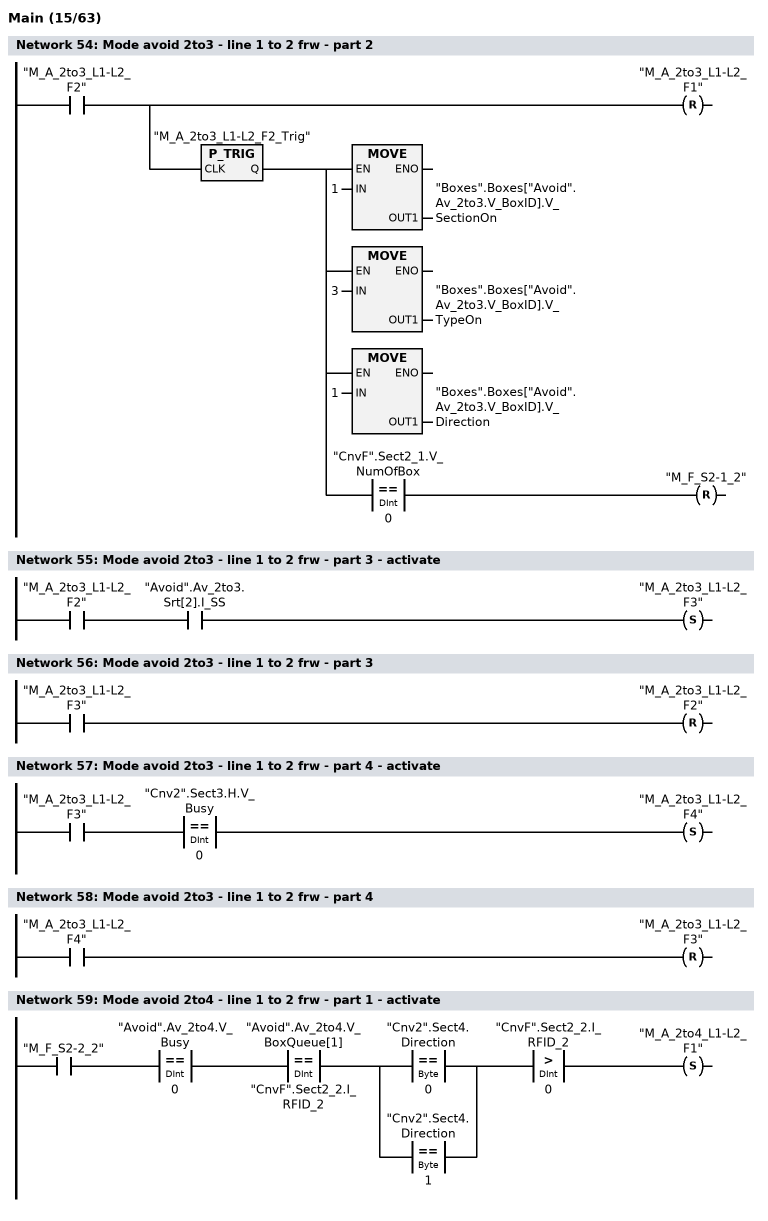
   RUNG wire#powerrail
      Contact( "M_A_2to3_L1-L2_F2" )
      wire#w1
      R_Coil( "M_A_2to3_L1-L2_F1" )
   END_RUNG
   RUNG wire#w1
      P_Trig( "M_A_2to3_L1-L2_F2_Trig" )
      wire#w2
      Move(in := 1, out1 => "Boxes".Boxes["Avoid".Av_2to3.V_BoxID].V_SectionOn)
   END_RUNG
   RUNG wire#w2
      Move(in := 3, out1 => "Boxes".Boxes["Avoid".Av_2to3.V_BoxID].V_TypeOn)
   END_RUNG
   RUNG wire#w2
      Move(in := 1, out1 => "Boxes".Boxes["Avoid".Av_2to3.V_BoxID].V_Direction)
   END_RUNG
   RUNG wire#w2
      { S7_Templates := "SrcType := DInt" } EQ_Contact(in1 := "CnvF".Sect2_1.V_NumOfBox, in2 := 0)
      R_Coil( "M_F_S2-1_2" )
   END_RUNG
   // the same network as SCL:
   IF "M_A_2to3_L1-L2_F2" THEN "M_A_2to3_L1-L2_F1" := FALSE; END_IF;
   #_w1 := "M_A_2to3_L1-L2_F2" AND NOT "M_A_2to3_L1-L2_F2_Trig";   // rising edge
   "M_A_2to3_L1-L2_F2_Trig" := "M_A_2to3_L1-L2_F2";
   IF #_w1 THEN
       "Boxes".Boxes["Avoid".Av_2to3.V_BoxID].V_SectionOn := 1;
       "Boxes".Boxes["Avoid".Av_2to3.V_BoxID].V_TypeOn := 3;
       "Boxes".Boxes["Avoid".Av_2to3.V_BoxID].V_Direction := 1;
   END_IF;
   IF #_w1 AND ("CnvF".Sect2_1.V_NumOfBox = 0) THEN "M_F_S2-1_2" := FALSE; END_IF;
END_REGION

REGION Network 55: Mode avoid 2to3 - line 1 to 2 frw - part 3 - activate
   RUNG wire#powerrail
      Contact( "M_A_2to3_L1-L2_F2" )
      Contact( "Avoid".Av_2to3.Srt[2].I_SS )
      S_Coil( "M_A_2to3_L1-L2_F3" )
   END_RUNG
   // the same network as SCL:
   IF "M_A_2to3_L1-L2_F2" AND "Avoid".Av_2to3.Srt[2].I_SS THEN "M_A_2to3_L1-L2_F3" := TRUE; END_IF;
END_REGION

REGION Network 56: Mode avoid 2to3 - line 1 to 2 frw - part 3
   RUNG wire#powerrail
      Contact( "M_A_2to3_L1-L2_F3" )
      R_Coil( "M_A_2to3_L1-L2_F2" )
   END_RUNG
   // the same network as SCL:
   IF "M_A_2to3_L1-L2_F3" THEN "M_A_2to3_L1-L2_F2" := FALSE; END_IF;
END_REGION

REGION Network 57: Mode avoid 2to3 - line 1 to 2 frw - part 4 - activate
   RUNG wire#powerrail
      Contact( "M_A_2to3_L1-L2_F3" )
      { S7_Templates := "SrcType := DInt" } EQ_Contact(in1 := "Cnv2".Sect3.H.V_Busy, in2 := 0)
      S_Coil( "M_A_2to3_L1-L2_F4" )
   END_RUNG
   // the same network as SCL:
   IF "M_A_2to3_L1-L2_F3" AND ("Cnv2".Sect3.H.V_Busy = 0) THEN "M_A_2to3_L1-L2_F4" := TRUE; END_IF;
END_REGION

REGION Network 58: Mode avoid 2to3 - line 1 to 2 frw - part 4
   RUNG wire#powerrail
      Contact( "M_A_2to3_L1-L2_F4" )
      R_Coil( "M_A_2to3_L1-L2_F3" )
   END_RUNG
   // the same network as SCL:
   IF "M_A_2to3_L1-L2_F4" THEN "M_A_2to3_L1-L2_F3" := FALSE; END_IF;
END_REGION

REGION Network 59: Mode avoid 2to4 - line 1 to 2 frw - part 1 - activate
   RUNG wire#powerrail
      Contact( "M_F_S2-2_2" )
      { S7_Templates := "SrcType := DInt" } EQ_Contact(in1 := "Avoid".Av_2to4.V_Busy, in2 := 0)
      { S7_Templates := "SrcType := DInt" } EQ_Contact(in1 := "Avoid".Av_2to4.V_BoxQueue[1], in2 := "CnvF".Sect2_2.I_RFID_2)
      wire#w1
      { S7_Templates := "SrcType := Byte" } EQ_Contact(in1 := "Cnv2".Sect4.Direction, in2 := 0)
      wire#w2
      { S7_Templates := "SrcType := DInt" } GT_Contact(in1 := "CnvF".Sect2_2.I_RFID_2, in2 := 0)
      S_Coil( "M_A_2to4_L1-L2_F1" )
   END_RUNG
   RUNG wire#w1
      { S7_Templates := "SrcType := Byte" } EQ_Contact(in1 := "Cnv2".Sect4.Direction, in2 := 1)
   END_RUNG wire#w2
   // the same network as SCL:
   IF "M_F_S2-2_2" AND ("Avoid".Av_2to4.V_Busy = 0) AND ("Avoid".Av_2to4.V_BoxQueue[1] = "CnvF".Sect2_2.I_RFID_2) AND (("Cnv2".Sect4.Direction = 0) OR ("Cnv2".Sect4.Direction = 1)) AND ("CnvF".Sect2_2.I_RFID_2 > 0) THEN
       "M_A_2to4_L1-L2_F1" := TRUE;
   END_IF;
END_REGION

REGION Network 60: Mode avoid 2to4 - line 1 to 2 frw - part 1
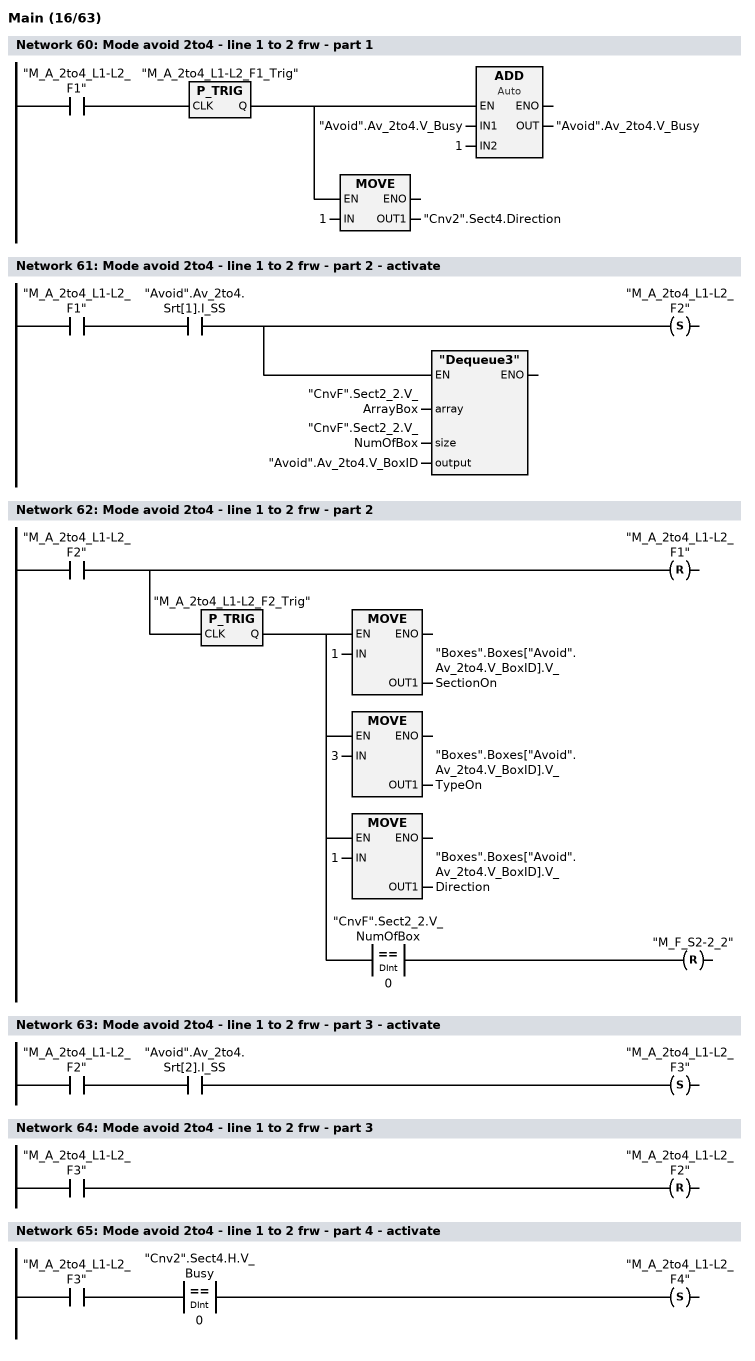
   RUNG wire#powerrail
      Contact( "M_A_2to4_L1-L2_F1" )
      P_Trig( "M_A_2to4_L1-L2_F1_Trig" )
      wire#w1
      Add(in1 := "Avoid".Av_2to4.V_Busy, in2 := 1, out => "Avoid".Av_2to4.V_Busy)
   END_RUNG
   RUNG wire#w1
      Move(in := 1, out1 => "Cnv2".Sect4.Direction)
   END_RUNG
   // the same network as SCL:
   #_w1 := "M_A_2to4_L1-L2_F1" AND NOT "M_A_2to4_L1-L2_F1_Trig";   // rising edge
   "M_A_2to4_L1-L2_F1_Trig" := "M_A_2to4_L1-L2_F1";
   IF #_w1 THEN
       "Avoid".Av_2to4.V_Busy := "Avoid".Av_2to4.V_Busy + 1;
       "Cnv2".Sect4.Direction := 1;
   END_IF;
END_REGION

REGION Network 61: Mode avoid 2to4 - line 1 to 2 frw - part 2 - activate
   RUNG wire#powerrail
      Contact( "M_A_2to4_L1-L2_F1" )
      Contact( "Avoid".Av_2to4.Srt[1].I_SS )
      wire#w1
      S_Coil( "M_A_2to4_L1-L2_F2" )
   END_RUNG
   RUNG wire#w1
      "Dequeue3"("array" := "CnvF".Sect2_2.V_ArrayBox, size := "CnvF".Sect2_2.V_NumOfBox, output := "Avoid".Av_2to4.V_BoxID)
   END_RUNG
   // the same network as SCL:
   IF "M_A_2to4_L1-L2_F1" AND "Avoid".Av_2to4.Srt[1].I_SS THEN
       "M_A_2to4_L1-L2_F2" := TRUE;
       "Dequeue3"("array" := "CnvF".Sect2_2.V_ArrayBox,
                  size := "CnvF".Sect2_2.V_NumOfBox,
                  output := "Avoid".Av_2to4.V_BoxID);
   END_IF;
END_REGION

REGION Network 62: Mode avoid 2to4 - line 1 to 2 frw - part 2
   RUNG wire#powerrail
      Contact( "M_A_2to4_L1-L2_F2" )
      wire#w1
      R_Coil( "M_A_2to4_L1-L2_F1" )
   END_RUNG
   RUNG wire#w1
      P_Trig( "M_A_2to4_L1-L2_F2_Trig" )
      wire#w2
      Move(in := 1, out1 => "Boxes".Boxes["Avoid".Av_2to4.V_BoxID].V_SectionOn)
   END_RUNG
   RUNG wire#w2
      Move(in := 3, out1 => "Boxes".Boxes["Avoid".Av_2to4.V_BoxID].V_TypeOn)
   END_RUNG
   RUNG wire#w2
      Move(in := 1, out1 => "Boxes".Boxes["Avoid".Av_2to4.V_BoxID].V_Direction)
   END_RUNG
   RUNG wire#w2
      { S7_Templates := "SrcType := DInt" } EQ_Contact(in1 := "CnvF".Sect2_2.V_NumOfBox, in2 := 0)
      R_Coil( "M_F_S2-2_2" )
   END_RUNG
   // the same network as SCL:
   IF "M_A_2to4_L1-L2_F2" THEN "M_A_2to4_L1-L2_F1" := FALSE; END_IF;
   #_w1 := "M_A_2to4_L1-L2_F2" AND NOT "M_A_2to4_L1-L2_F2_Trig";   // rising edge
   "M_A_2to4_L1-L2_F2_Trig" := "M_A_2to4_L1-L2_F2";
   IF #_w1 THEN
       "Boxes".Boxes["Avoid".Av_2to4.V_BoxID].V_SectionOn := 1;
       "Boxes".Boxes["Avoid".Av_2to4.V_BoxID].V_TypeOn := 3;
       "Boxes".Boxes["Avoid".Av_2to4.V_BoxID].V_Direction := 1;
   END_IF;
   IF #_w1 AND ("CnvF".Sect2_2.V_NumOfBox = 0) THEN "M_F_S2-2_2" := FALSE; END_IF;
END_REGION

REGION Network 63: Mode avoid 2to4 - line 1 to 2 frw - part 3 - activate
   RUNG wire#powerrail
      Contact( "M_A_2to4_L1-L2_F2" )
      Contact( "Avoid".Av_2to4.Srt[2].I_SS )
      S_Coil( "M_A_2to4_L1-L2_F3" )
   END_RUNG
   // the same network as SCL:
   IF "M_A_2to4_L1-L2_F2" AND "Avoid".Av_2to4.Srt[2].I_SS THEN "M_A_2to4_L1-L2_F3" := TRUE; END_IF;
END_REGION

REGION Network 64: Mode avoid 2to4 - line 1 to 2 frw - part 3
   RUNG wire#powerrail
      Contact( "M_A_2to4_L1-L2_F3" )
      R_Coil( "M_A_2to4_L1-L2_F2" )
   END_RUNG
   // the same network as SCL:
   IF "M_A_2to4_L1-L2_F3" THEN "M_A_2to4_L1-L2_F2" := FALSE; END_IF;
END_REGION

REGION Network 65: Mode avoid 2to4 - line 1 to 2 frw - part 4 - activate
   RUNG wire#powerrail
      Contact( "M_A_2to4_L1-L2_F3" )
      { S7_Templates := "SrcType := DInt" } EQ_Contact(in1 := "Cnv2".Sect4.H.V_Busy, in2 := 0)
      S_Coil( "M_A_2to4_L1-L2_F4" )
   END_RUNG
   // the same network as SCL:
   IF "M_A_2to4_L1-L2_F3" AND ("Cnv2".Sect4.H.V_Busy = 0) THEN "M_A_2to4_L1-L2_F4" := TRUE; END_IF;
END_REGION

REGION Network 66: Mode avoid 2to4 - line 1 to 2 frw - part 4
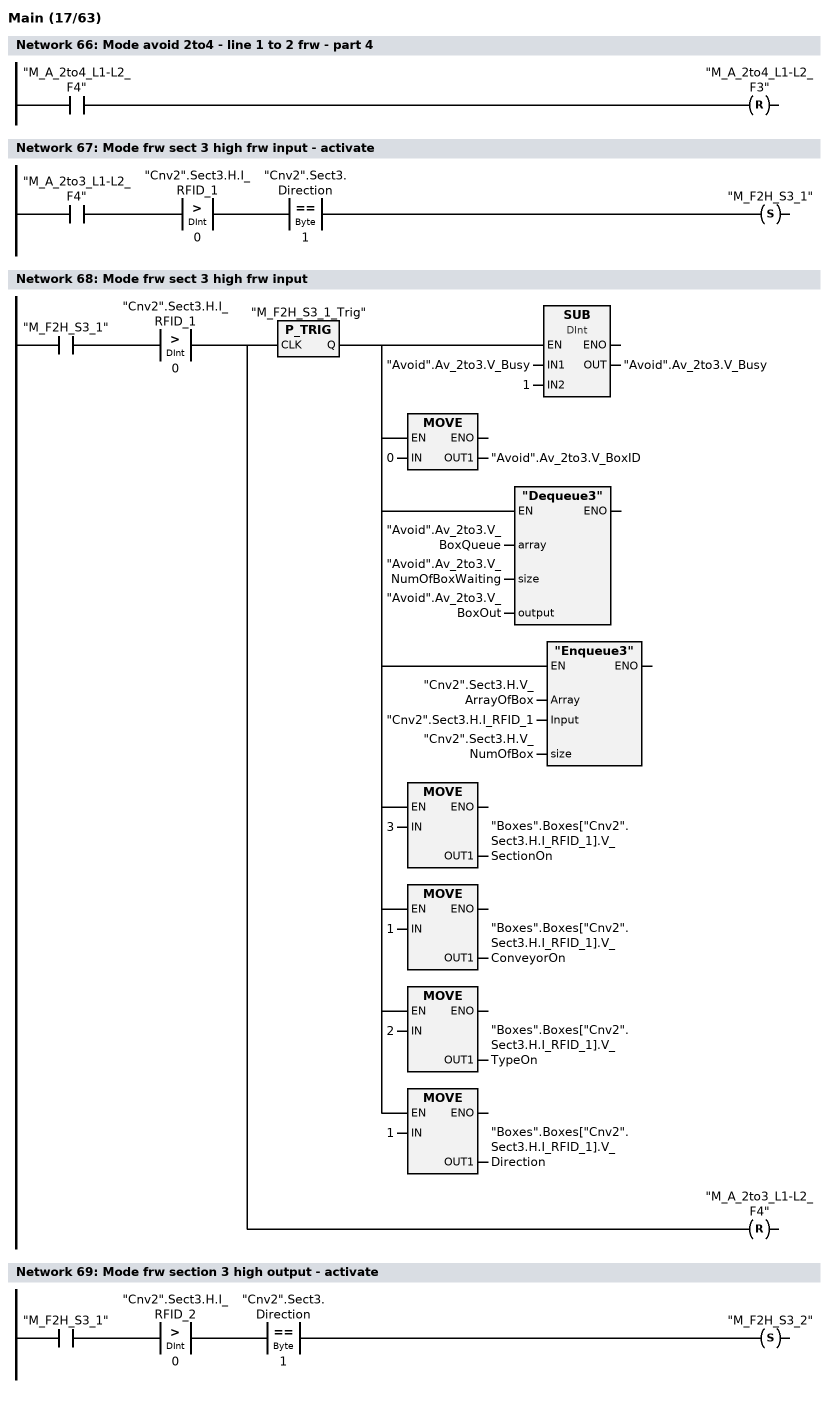
   RUNG wire#powerrail
      Contact( "M_A_2to4_L1-L2_F4" )
      R_Coil( "M_A_2to4_L1-L2_F3" )
   END_RUNG
   // the same network as SCL:
   IF "M_A_2to4_L1-L2_F4" THEN "M_A_2to4_L1-L2_F3" := FALSE; END_IF;
END_REGION

REGION Network 67: Mode frw sect 3 high frw input - activate
   RUNG wire#powerrail
      Contact( "M_A_2to3_L1-L2_F4" )
      { S7_Templates := "SrcType := DInt" } GT_Contact(in1 := "Cnv2".Sect3.H.I_RFID_1, in2 := 0)
      { S7_Templates := "SrcType := Byte" } EQ_Contact(in1 := "Cnv2".Sect3.Direction, in2 := 1)
      S_Coil( "M_F2H_S3_1" )
   END_RUNG
   // the same network as SCL:
   IF "M_A_2to3_L1-L2_F4" AND ("Cnv2".Sect3.H.I_RFID_1 > 0) AND ("Cnv2".Sect3.Direction = 1) THEN
       "M_F2H_S3_1" := TRUE;
   END_IF;
END_REGION

REGION Network 68: Mode frw sect 3 high frw input
   RUNG wire#powerrail
      Contact( "M_F2H_S3_1" )
      { S7_Templates := "SrcType := DInt" } GT_Contact(in1 := "Cnv2".Sect3.H.I_RFID_1, in2 := 0)
      wire#w1
      P_Trig( "M_F2H_S3_1_Trig" )
      wire#w2
      { S7_Templates := "SrcType := DInt" } Sub(in1 := "Avoid".Av_2to3.V_Busy, in2 := 1, out => "Avoid".Av_2to3.V_Busy)
   END_RUNG
   RUNG wire#w2
      Move(in := 0, out1 => "Avoid".Av_2to3.V_BoxID)
   END_RUNG
   RUNG wire#w2
      "Dequeue3"("array" := "Avoid".Av_2to3.V_BoxQueue, size := "Avoid".Av_2to3.V_NumOfBoxWaiting, output := "Avoid".Av_2to3.V_BoxOut)
   END_RUNG
   RUNG wire#w2
      "Enqueue3"("Array" := "Cnv2".Sect3.H.V_ArrayOfBox, Input := "Cnv2".Sect3.H.I_RFID_1, size := "Cnv2".Sect3.H.V_NumOfBox)
   END_RUNG
   RUNG wire#w2
      Move(in := 3, out1 => "Boxes".Boxes["Cnv2".Sect3.H.I_RFID_1].V_SectionOn)
   END_RUNG
   RUNG wire#w2
      Move(in := 1, out1 => "Boxes".Boxes["Cnv2".Sect3.H.I_RFID_1].V_ConveyorOn)
   END_RUNG
   RUNG wire#w2
      Move(in := 2, out1 => "Boxes".Boxes["Cnv2".Sect3.H.I_RFID_1].V_TypeOn)
   END_RUNG
   RUNG wire#w2
      Move(in := 1, out1 => "Boxes".Boxes["Cnv2".Sect3.H.I_RFID_1].V_Direction)
   END_RUNG
   RUNG wire#w1
      R_Coil( "M_A_2to3_L1-L2_F4" )
   END_RUNG
   // the same network as SCL:
   #_w1 := "M_F2H_S3_1" AND ("Cnv2".Sect3.H.I_RFID_1 > 0);
   #_w2 := #_w1 AND NOT "M_F2H_S3_1_Trig";   // rising edge
   "M_F2H_S3_1_Trig" := #_w1;
   IF #_w2 THEN
       "Avoid".Av_2to3.V_Busy := "Avoid".Av_2to3.V_Busy - 1;
       "Avoid".Av_2to3.V_BoxID := 0;
       "Dequeue3"("array" := "Avoid".Av_2to3.V_BoxQueue,
                  size := "Avoid".Av_2to3.V_NumOfBoxWaiting,
                  output := "Avoid".Av_2to3.V_BoxOut);
       "Enqueue3"("Array" := "Cnv2".Sect3.H.V_ArrayOfBox,
                  Input := "Cnv2".Sect3.H.I_RFID_1,
                  size := "Cnv2".Sect3.H.V_NumOfBox);
       "Boxes".Boxes["Cnv2".Sect3.H.I_RFID_1].V_SectionOn := 3;
       "Boxes".Boxes["Cnv2".Sect3.H.I_RFID_1].V_ConveyorOn := 1;
       "Boxes".Boxes["Cnv2".Sect3.H.I_RFID_1].V_TypeOn := 2;
       "Boxes".Boxes["Cnv2".Sect3.H.I_RFID_1].V_Direction := 1;
   END_IF;
   IF #_w1 THEN "M_A_2to3_L1-L2_F4" := FALSE; END_IF;
END_REGION

REGION Network 69: Mode frw section 3 high output - activate
   RUNG wire#powerrail
      Contact( "M_F2H_S3_1" )
      { S7_Templates := "SrcType := DInt" } GT_Contact(in1 := "Cnv2".Sect3.H.I_RFID_2, in2 := 0)
      { S7_Templates := "SrcType := Byte" } EQ_Contact(in1 := "Cnv2".Sect3.Direction, in2 := 1)
      S_Coil( "M_F2H_S3_2" )
   END_RUNG
   // the same network as SCL:
   IF "M_F2H_S3_1" AND ("Cnv2".Sect3.H.I_RFID_2 > 0) AND ("Cnv2".Sect3.Direction = 1) THEN
       "M_F2H_S3_2" := TRUE;
   END_IF;
END_REGION

REGION Network 70: Mode frw section 3 high output
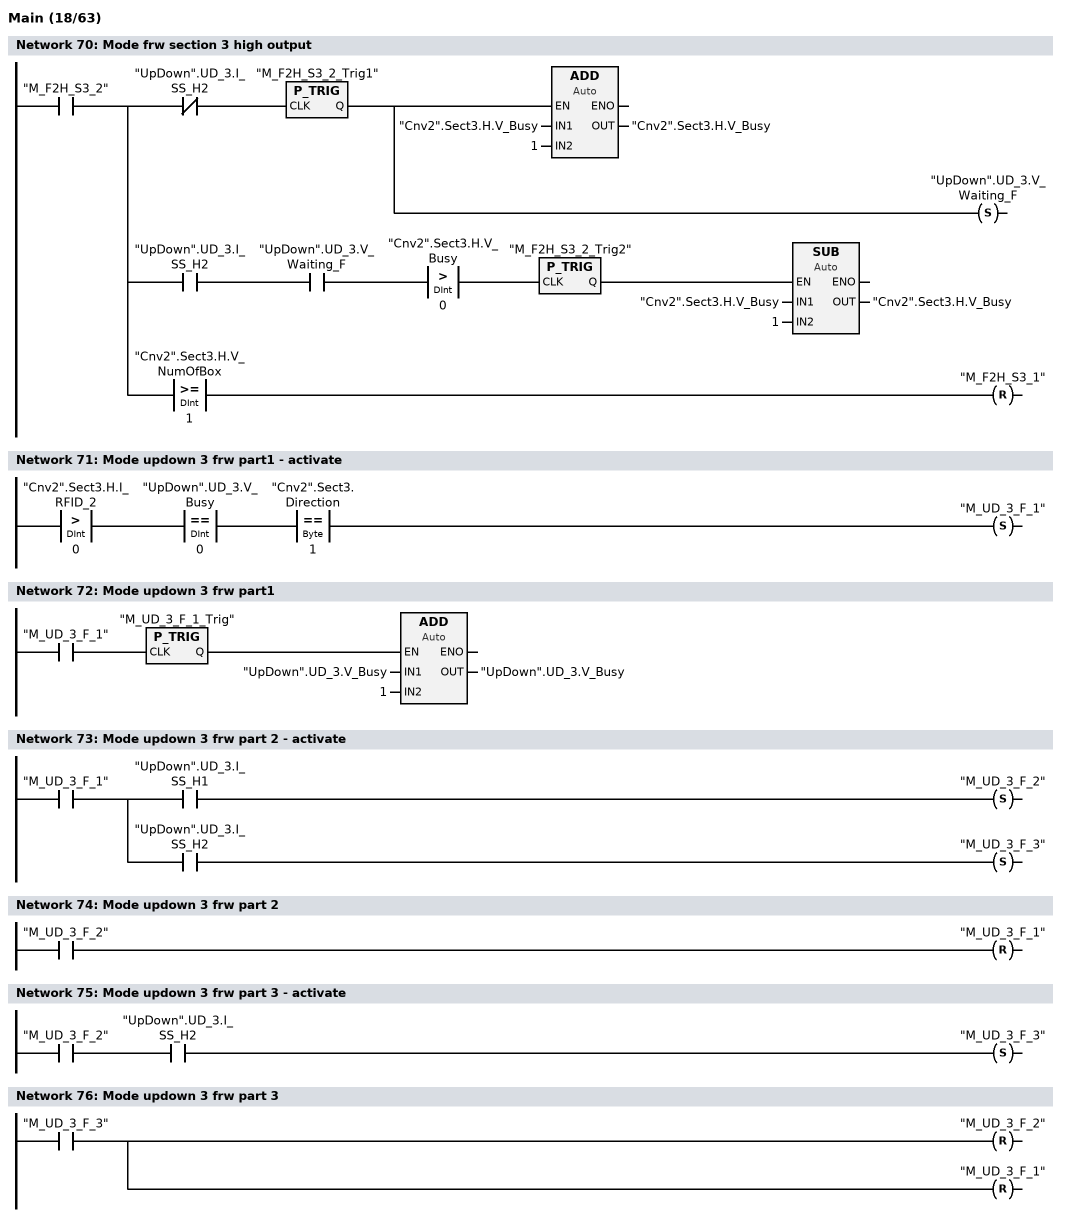
   RUNG wire#powerrail
      Contact( "M_F2H_S3_2" )
      wire#w1
      I_Contact( "UpDown".UD_3.I_SS_H2 )
      P_Trig( "M_F2H_S3_2_Trig1" )
      wire#w2
      Add(in1 := "Cnv2".Sect3.H.V_Busy, in2 := 1, out => "Cnv2".Sect3.H.V_Busy)
   END_RUNG
   RUNG wire#w2
      S_Coil( "UpDown".UD_3.V_Waiting_F )
   END_RUNG
   RUNG wire#w1
      Contact( "UpDown".UD_3.I_SS_H2 )
      Contact( "UpDown".UD_3.V_Waiting_F )
      { S7_Templates := "SrcType := DInt" } GT_Contact(in1 := "Cnv2".Sect3.H.V_Busy, in2 := 0)
      P_Trig( "M_F2H_S3_2_Trig2" )
      Sub(in1 := "Cnv2".Sect3.H.V_Busy, in2 := 1, out => "Cnv2".Sect3.H.V_Busy)
   END_RUNG
   RUNG wire#w1
      { S7_Templates := "SrcType := DInt" } GE_Contact(in1 := "Cnv2".Sect3.H.V_NumOfBox, in2 := 1)
      R_Coil( "M_F2H_S3_1" )
   END_RUNG
   // the same network as SCL:
   #_w1 := "M_F2H_S3_2" AND NOT "UpDown".UD_3.I_SS_H2;
   #_w2 := #_w1 AND NOT "M_F2H_S3_2_Trig1";   // rising edge
   "M_F2H_S3_2_Trig1" := #_w1;
   IF #_w2 THEN
       "Cnv2".Sect3.H.V_Busy := "Cnv2".Sect3.H.V_Busy + 1;
       "UpDown".UD_3.V_Waiting_F := TRUE;
   END_IF;
   #_w3 := "M_F2H_S3_2" AND "UpDown".UD_3.I_SS_H2 AND "UpDown".UD_3.V_Waiting_F AND ("Cnv2".Sect3.H.V_Busy > 0);
   #_w4 := #_w3 AND NOT "M_F2H_S3_2_Trig2";   // rising edge
   "M_F2H_S3_2_Trig2" := #_w3;
   IF #_w4 THEN "Cnv2".Sect3.H.V_Busy := "Cnv2".Sect3.H.V_Busy - 1; END_IF;
   IF "M_F2H_S3_2" AND ("Cnv2".Sect3.H.V_NumOfBox >= 1) THEN "M_F2H_S3_1" := FALSE; END_IF;
END_REGION

REGION Network 71: Mode updown 3 frw part1 - activate
   RUNG wire#powerrail
      { S7_Templates := "SrcType := DInt" } GT_Contact(in1 := "Cnv2".Sect3.H.I_RFID_2, in2 := 0)
      { S7_Templates := "SrcType := DInt" } EQ_Contact(in1 := "UpDown".UD_3.V_Busy, in2 := 0)
      { S7_Templates := "SrcType := Byte" } EQ_Contact(in1 := "Cnv2".Sect3.Direction, in2 := 1)
      S_Coil( "M_UD_3_F_1" )
   END_RUNG
   // the same network as SCL:
   IF ("Cnv2".Sect3.H.I_RFID_2 > 0) AND ("UpDown".UD_3.V_Busy = 0) AND ("Cnv2".Sect3.Direction = 1) THEN
       "M_UD_3_F_1" := TRUE;
   END_IF;
END_REGION

REGION Network 72: Mode updown 3 frw part1
   RUNG wire#powerrail
      Contact( "M_UD_3_F_1" )
      P_Trig( "M_UD_3_F_1_Trig" )
      Add(in1 := "UpDown".UD_3.V_Busy, in2 := 1, out => "UpDown".UD_3.V_Busy)
   END_RUNG
   // the same network as SCL:
   #_w1 := "M_UD_3_F_1" AND NOT "M_UD_3_F_1_Trig";   // rising edge
   "M_UD_3_F_1_Trig" := "M_UD_3_F_1";
   IF #_w1 THEN "UpDown".UD_3.V_Busy := "UpDown".UD_3.V_Busy + 1; END_IF;
END_REGION

REGION Network 73: Mode updown 3 frw part 2 - activate
   RUNG wire#powerrail
      Contact( "M_UD_3_F_1" )
      wire#w1
      Contact( "UpDown".UD_3.I_SS_H1 )
      S_Coil( "M_UD_3_F_2" )
   END_RUNG
   RUNG wire#w1
      Contact( "UpDown".UD_3.I_SS_H2 )
      S_Coil( "M_UD_3_F_3" )
   END_RUNG
   // the same network as SCL:
   IF "M_UD_3_F_1" AND "UpDown".UD_3.I_SS_H1 THEN "M_UD_3_F_2" := TRUE; END_IF;
   IF "M_UD_3_F_1" AND "UpDown".UD_3.I_SS_H2 THEN "M_UD_3_F_3" := TRUE; END_IF;
END_REGION

REGION Network 74: Mode updown 3 frw part 2
   RUNG wire#powerrail
      Contact( "M_UD_3_F_2" )
      R_Coil( "M_UD_3_F_1" )
   END_RUNG
   // the same network as SCL:
   IF "M_UD_3_F_2" THEN "M_UD_3_F_1" := FALSE; END_IF;
END_REGION

REGION Network 75: Mode updown 3 frw part 3 - activate
   RUNG wire#powerrail
      Contact( "M_UD_3_F_2" )
      Contact( "UpDown".UD_3.I_SS_H2 )
      S_Coil( "M_UD_3_F_3" )
   END_RUNG
   // the same network as SCL:
   IF "M_UD_3_F_2" AND "UpDown".UD_3.I_SS_H2 THEN "M_UD_3_F_3" := TRUE; END_IF;
END_REGION

REGION Network 76: Mode updown 3 frw part 3
   RUNG wire#powerrail
      Contact( "M_UD_3_F_3" )
      wire#w1
      R_Coil( "M_UD_3_F_2" )
   END_RUNG
   RUNG wire#w1
      R_Coil( "M_UD_3_F_1" )
   END_RUNG
   // the same network as SCL:
   IF "M_UD_3_F_3" THEN
       "M_UD_3_F_2" := FALSE;
       "M_UD_3_F_1" := FALSE;
   END_IF;
END_REGION

REGION Network 77: Mode updown 3 frw part 4 - activate
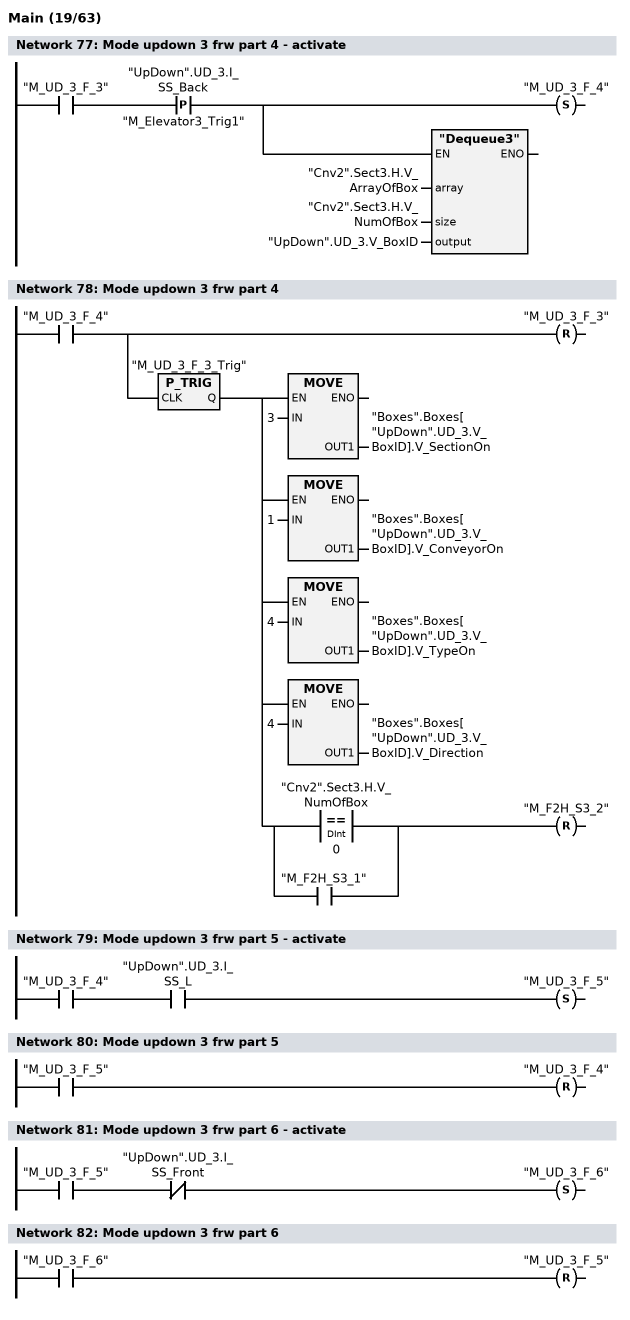
   RUNG wire#powerrail
      Contact( "M_UD_3_F_3" )
      P_Contact(operand := "UpDown".UD_3.I_SS_Back, bit := "M_Elevator3_Trig1")
      wire#w1
      S_Coil( "M_UD_3_F_4" )
   END_RUNG
   RUNG wire#w1
      "Dequeue3"("array" := "Cnv2".Sect3.H.V_ArrayOfBox, size := "Cnv2".Sect3.H.V_NumOfBox, output := "UpDown".UD_3.V_BoxID)
   END_RUNG
   // the same network as SCL:
   #_w1 := "M_UD_3_F_3" AND "UpDown".UD_3.I_SS_Back AND NOT "M_Elevator3_Trig1";   // rising edge of "UpDown".UD_3.I_SS_Back
   "M_Elevator3_Trig1" := "UpDown".UD_3.I_SS_Back;
   IF #_w1 THEN
       "M_UD_3_F_4" := TRUE;
       "Dequeue3"("array" := "Cnv2".Sect3.H.V_ArrayOfBox,
                  size := "Cnv2".Sect3.H.V_NumOfBox,
                  output := "UpDown".UD_3.V_BoxID);
   END_IF;
END_REGION

REGION Network 78: Mode updown 3 frw part 4
   RUNG wire#powerrail
      Contact( "M_UD_3_F_4" )
      wire#w1
      R_Coil( "M_UD_3_F_3" )
   END_RUNG
   RUNG wire#w1
      P_Trig( "M_UD_3_F_3_Trig" )
      wire#w2
      Move(in := 3, out1 => "Boxes".Boxes["UpDown".UD_3.V_BoxID].V_SectionOn)
   END_RUNG
   RUNG wire#w2
      Move(in := 1, out1 => "Boxes".Boxes["UpDown".UD_3.V_BoxID].V_ConveyorOn)
   END_RUNG
   RUNG wire#w2
      Move(in := 4, out1 => "Boxes".Boxes["UpDown".UD_3.V_BoxID].V_TypeOn)
   END_RUNG
   RUNG wire#w2
      Move(in := 4, out1 => "Boxes".Boxes["UpDown".UD_3.V_BoxID].V_Direction)
   END_RUNG
   RUNG wire#w2
      { S7_Templates := "SrcType := DInt" } EQ_Contact(in1 := "Cnv2".Sect3.H.V_NumOfBox, in2 := 0)
      wire#w3
      R_Coil( "M_F2H_S3_2" )
   END_RUNG
   RUNG wire#w2
      Contact( "M_F2H_S3_1" )
   END_RUNG wire#w3
   // the same network as SCL:
   IF "M_UD_3_F_4" THEN "M_UD_3_F_3" := FALSE; END_IF;
   #_w1 := "M_UD_3_F_4" AND NOT "M_UD_3_F_3_Trig";   // rising edge
   "M_UD_3_F_3_Trig" := "M_UD_3_F_4";
   IF #_w1 THEN
       "Boxes".Boxes["UpDown".UD_3.V_BoxID].V_SectionOn := 3;
       "Boxes".Boxes["UpDown".UD_3.V_BoxID].V_ConveyorOn := 1;
       "Boxes".Boxes["UpDown".UD_3.V_BoxID].V_TypeOn := 4;
       "Boxes".Boxes["UpDown".UD_3.V_BoxID].V_Direction := 4;
   END_IF;
   IF #_w1 AND (("Cnv2".Sect3.H.V_NumOfBox = 0) OR "M_F2H_S3_1") THEN "M_F2H_S3_2" := FALSE; END_IF;
END_REGION

REGION Network 79: Mode updown 3 frw part 5 - activate
   RUNG wire#powerrail
      Contact( "M_UD_3_F_4" )
      Contact( "UpDown".UD_3.I_SS_L )
      S_Coil( "M_UD_3_F_5" )
   END_RUNG
   // the same network as SCL:
   IF "M_UD_3_F_4" AND "UpDown".UD_3.I_SS_L THEN "M_UD_3_F_5" := TRUE; END_IF;
END_REGION

REGION Network 80: Mode updown 3 frw part 5
   RUNG wire#powerrail
      Contact( "M_UD_3_F_5" )
      R_Coil( "M_UD_3_F_4" )
   END_RUNG
   // the same network as SCL:
   IF "M_UD_3_F_5" THEN "M_UD_3_F_4" := FALSE; END_IF;
END_REGION

REGION Network 81: Mode updown 3 frw part 6 - activate
   RUNG wire#powerrail
      Contact( "M_UD_3_F_5" )
      I_Contact( "UpDown".UD_3.I_SS_Front )
      S_Coil( "M_UD_3_F_6" )
   END_RUNG
   // the same network as SCL:
   IF "M_UD_3_F_5" AND NOT "UpDown".UD_3.I_SS_Front THEN "M_UD_3_F_6" := TRUE; END_IF;
END_REGION

REGION Network 82: Mode updown 3 frw part 6
   RUNG wire#powerrail
      Contact( "M_UD_3_F_6" )
      R_Coil( "M_UD_3_F_5" )
   END_RUNG
   // the same network as SCL:
   IF "M_UD_3_F_6" THEN "M_UD_3_F_5" := FALSE; END_IF;
END_REGION

REGION Network 83: Mode updown 3 frw part 7 - activate
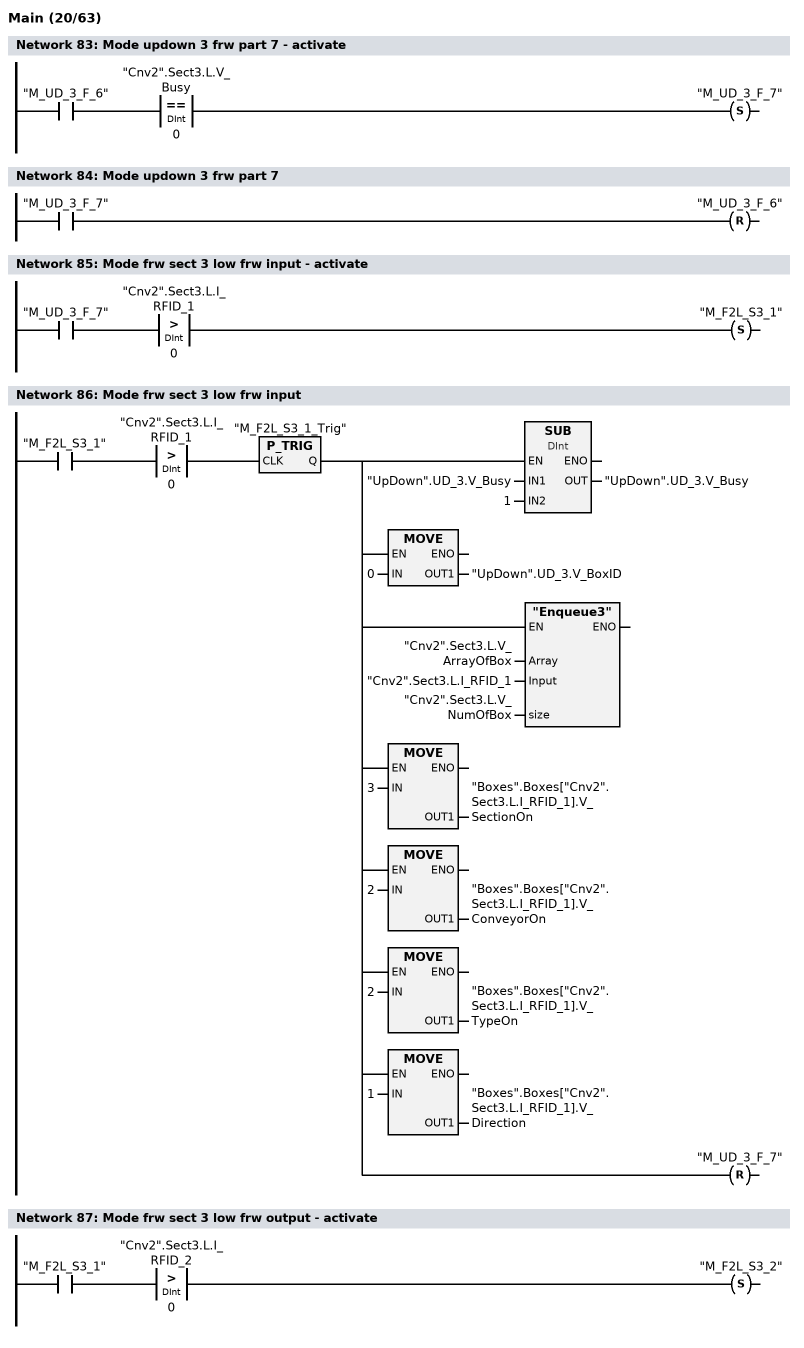
   RUNG wire#powerrail
      Contact( "M_UD_3_F_6" )
      { S7_Templates := "SrcType := DInt" } EQ_Contact(in1 := "Cnv2".Sect3.L.V_Busy, in2 := 0)
      S_Coil( "M_UD_3_F_7" )
   END_RUNG
   // the same network as SCL:
   IF "M_UD_3_F_6" AND ("Cnv2".Sect3.L.V_Busy = 0) THEN "M_UD_3_F_7" := TRUE; END_IF;
END_REGION

REGION Network 84: Mode updown 3 frw part 7
   RUNG wire#powerrail
      Contact( "M_UD_3_F_7" )
      R_Coil( "M_UD_3_F_6" )
   END_RUNG
   // the same network as SCL:
   IF "M_UD_3_F_7" THEN "M_UD_3_F_6" := FALSE; END_IF;
END_REGION

REGION Network 85: Mode frw sect 3 low frw input - activate
   RUNG wire#powerrail
      Contact( "M_UD_3_F_7" )
      { S7_Templates := "SrcType := DInt" } GT_Contact(in1 := "Cnv2".Sect3.L.I_RFID_1, in2 := 0)
      S_Coil( "M_F2L_S3_1" )
   END_RUNG
   // the same network as SCL:
   IF "M_UD_3_F_7" AND ("Cnv2".Sect3.L.I_RFID_1 > 0) THEN "M_F2L_S3_1" := TRUE; END_IF;
END_REGION

REGION Network 86: Mode frw sect 3 low frw input
   RUNG wire#powerrail
      Contact( "M_F2L_S3_1" )
      { S7_Templates := "SrcType := DInt" } GT_Contact(in1 := "Cnv2".Sect3.L.I_RFID_1, in2 := 0)
      P_Trig( "M_F2L_S3_1_Trig" )
      wire#w1
      { S7_Templates := "SrcType := DInt" } Sub(in1 := "UpDown".UD_3.V_Busy, in2 := 1, out => "UpDown".UD_3.V_Busy)
   END_RUNG
   RUNG wire#w1
      Move(in := 0, out1 => "UpDown".UD_3.V_BoxID)
   END_RUNG
   RUNG wire#w1
      "Enqueue3"("Array" := "Cnv2".Sect3.L.V_ArrayOfBox, Input := "Cnv2".Sect3.L.I_RFID_1, size := "Cnv2".Sect3.L.V_NumOfBox)
   END_RUNG
   RUNG wire#w1
      Move(in := 3, out1 => "Boxes".Boxes["Cnv2".Sect3.L.I_RFID_1].V_SectionOn)
   END_RUNG
   RUNG wire#w1
      Move(in := 2, out1 => "Boxes".Boxes["Cnv2".Sect3.L.I_RFID_1].V_ConveyorOn)
   END_RUNG
   RUNG wire#w1
      Move(in := 2, out1 => "Boxes".Boxes["Cnv2".Sect3.L.I_RFID_1].V_TypeOn)
   END_RUNG
   RUNG wire#w1
      Move(in := 1, out1 => "Boxes".Boxes["Cnv2".Sect3.L.I_RFID_1].V_Direction)
   END_RUNG
   RUNG wire#w1
      R_Coil( "M_UD_3_F_7" )
   END_RUNG
   // the same network as SCL:
   #_w1 := "M_F2L_S3_1" AND ("Cnv2".Sect3.L.I_RFID_1 > 0);
   #_w2 := #_w1 AND NOT "M_F2L_S3_1_Trig";   // rising edge
   "M_F2L_S3_1_Trig" := #_w1;
   IF #_w2 THEN
       "UpDown".UD_3.V_Busy := "UpDown".UD_3.V_Busy - 1;
       "UpDown".UD_3.V_BoxID := 0;
       "Enqueue3"("Array" := "Cnv2".Sect3.L.V_ArrayOfBox,
                  Input := "Cnv2".Sect3.L.I_RFID_1,
                  size := "Cnv2".Sect3.L.V_NumOfBox);
       "Boxes".Boxes["Cnv2".Sect3.L.I_RFID_1].V_SectionOn := 3;
       "Boxes".Boxes["Cnv2".Sect3.L.I_RFID_1].V_ConveyorOn := 2;
       "Boxes".Boxes["Cnv2".Sect3.L.I_RFID_1].V_TypeOn := 2;
       "Boxes".Boxes["Cnv2".Sect3.L.I_RFID_1].V_Direction := 1;
       "M_UD_3_F_7" := FALSE;
   END_IF;
END_REGION

REGION Network 87: Mode frw sect 3 low frw output - activate
   RUNG wire#powerrail
      Contact( "M_F2L_S3_1" )
      { S7_Templates := "SrcType := DInt" } GT_Contact(in1 := "Cnv2".Sect3.L.I_RFID_2, in2 := 0)
      S_Coil( "M_F2L_S3_2" )
   END_RUNG
   // the same network as SCL:
   IF "M_F2L_S3_1" AND ("Cnv2".Sect3.L.I_RFID_2 > 0) THEN "M_F2L_S3_2" := TRUE; END_IF;
END_REGION

REGION Network 88: Mode frw sect 3 low frw output
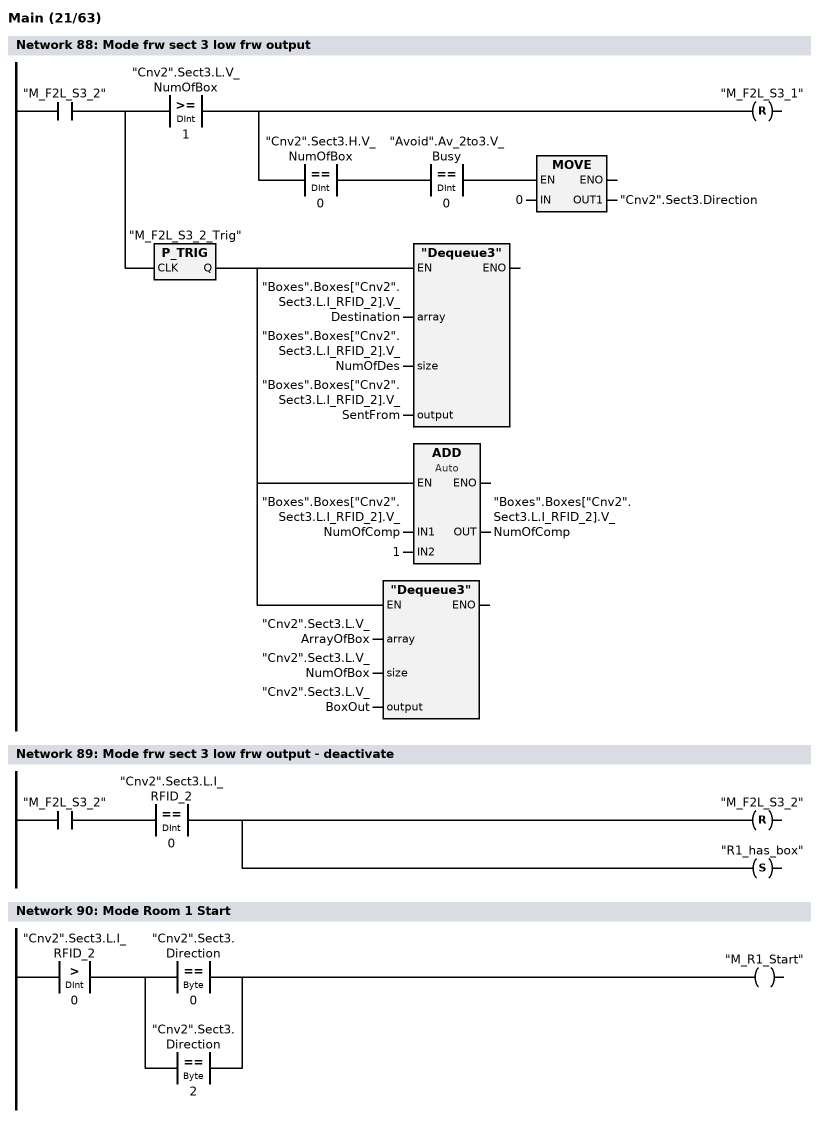
   RUNG wire#powerrail
      Contact( "M_F2L_S3_2" )
      wire#w1
      { S7_Templates := "SrcType := DInt" } GE_Contact(in1 := "Cnv2".Sect3.L.V_NumOfBox, in2 := 1)
      wire#w2
      R_Coil( "M_F2L_S3_1" )
   END_RUNG
   RUNG wire#w2
      { S7_Templates := "SrcType := DInt" } EQ_Contact(in1 := "Cnv2".Sect3.H.V_NumOfBox, in2 := 0)
      { S7_Templates := "SrcType := DInt" } EQ_Contact(in1 := "Avoid".Av_2to3.V_Busy, in2 := 0)
      Move(in := 0, out1 => "Cnv2".Sect3.Direction)
   END_RUNG
   RUNG wire#w1
      P_Trig( "M_F2L_S3_2_Trig" )
      wire#w3
      "Dequeue3"("array" := "Boxes".Boxes["Cnv2".Sect3.L.I_RFID_2].V_Destination, size := "Boxes".Boxes["Cnv2".Sect3.L.I_RFID_2].V_NumOfDes, output := "Boxes".Boxes["Cnv2".Sect3.L.I_RFID_2].V_SentFrom)
   END_RUNG
   RUNG wire#w3
      Add(in1 := "Boxes".Boxes["Cnv2".Sect3.L.I_RFID_2].V_NumOfComp, in2 := 1, out => "Boxes".Boxes["Cnv2".Sect3.L.I_RFID_2].V_NumOfComp)
   END_RUNG
   RUNG wire#w3
      "Dequeue3"("array" := "Cnv2".Sect3.L.V_ArrayOfBox, size := "Cnv2".Sect3.L.V_NumOfBox, output := "Cnv2".Sect3.L.V_BoxOut)
   END_RUNG
   // the same network as SCL:
   #_w1 := "M_F2L_S3_2" AND ("Cnv2".Sect3.L.V_NumOfBox >= 1);
   IF #_w1 THEN "M_F2L_S3_1" := FALSE; END_IF;
   IF #_w1 AND ("Cnv2".Sect3.H.V_NumOfBox = 0) AND ("Avoid".Av_2to3.V_Busy = 0) THEN
       "Cnv2".Sect3.Direction := 0;
   END_IF;
   #_w2 := "M_F2L_S3_2" AND NOT "M_F2L_S3_2_Trig";   // rising edge
   "M_F2L_S3_2_Trig" := "M_F2L_S3_2";
   IF #_w2 THEN
       "Dequeue3"("array" := "Boxes".Boxes["Cnv2".Sect3.L.I_RFID_2].V_Destination,
                  size := "Boxes".Boxes["Cnv2".Sect3.L.I_RFID_2].V_NumOfDes,
                  output := "Boxes".Boxes["Cnv2".Sect3.L.I_RFID_2].V_SentFrom);
       "Boxes".Boxes["Cnv2".Sect3.L.I_RFID_2].V_NumOfComp := "Boxes".Boxes["Cnv2".Sect3.L.I_RFID_2].V_NumOfComp + 1;
       "Dequeue3"("array" := "Cnv2".Sect3.L.V_ArrayOfBox,
                  size := "Cnv2".Sect3.L.V_NumOfBox,
                  output := "Cnv2".Sect3.L.V_BoxOut);
   END_IF;
END_REGION

REGION Network 89: Mode frw sect 3 low frw output - deactivate
   RUNG wire#powerrail
      Contact( "M_F2L_S3_2" )
      { S7_Templates := "SrcType := DInt" } EQ_Contact(in1 := "Cnv2".Sect3.L.I_RFID_2, in2 := 0)
      wire#w1
      R_Coil( "M_F2L_S3_2" )
   END_RUNG
   RUNG wire#w1
      S_Coil( "R1_has_box" )
   END_RUNG
   // the same network as SCL:
   #_w1 := "M_F2L_S3_2" AND ("Cnv2".Sect3.L.I_RFID_2 = 0);
   IF #_w1 THEN
       "M_F2L_S3_2" := FALSE;
       "R1_has_box" := TRUE;
   END_IF;
END_REGION

REGION Network 90: Mode Room 1 Start
   RUNG wire#powerrail
      { S7_Templates := "SrcType := DInt" } GT_Contact(in1 := "Cnv2".Sect3.L.I_RFID_2, in2 := 0)
      wire#w1
      { S7_Templates := "SrcType := Byte" } EQ_Contact(in1 := "Cnv2".Sect3.Direction, in2 := 0)
      wire#w2
      Coil( "M_R1_Start" )
   END_RUNG
   RUNG wire#w1
      { S7_Templates := "SrcType := Byte" } EQ_Contact(in1 := "Cnv2".Sect3.Direction, in2 := 2)
   END_RUNG wire#w2
   // the same network as SCL:
   "M_R1_Start" := ("Cnv2".Sect3.L.I_RFID_2 > 0) AND (("Cnv2".Sect3.Direction = 0) OR ("Cnv2".Sect3.Direction = 2));
END_REGION

REGION Network 91: Mode Room 1 - choose return or continue and Mode back sect 3 input - activate
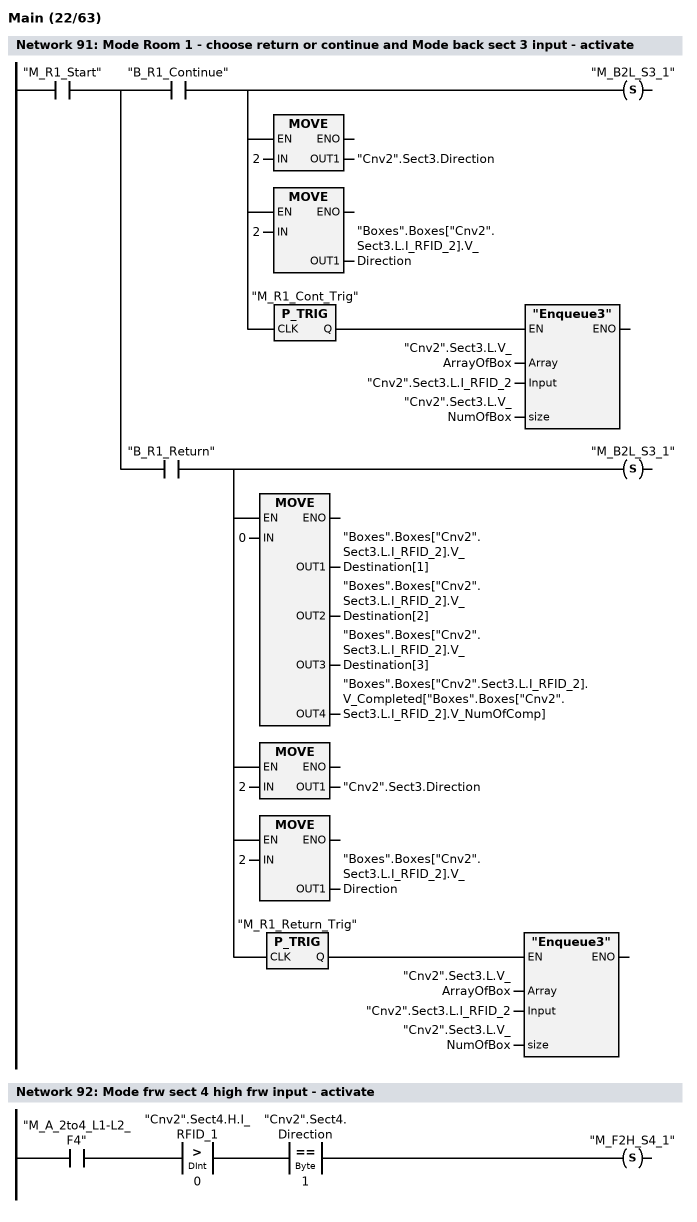
   RUNG wire#powerrail
      Contact( "M_R1_Start" )
      wire#w1
      Contact( "B_R1_Continue" )
      wire#w2
      S_Coil( "M_B2L_S3_1" )
   END_RUNG
   RUNG wire#w2
      Move(in := 2, out1 => "Cnv2".Sect3.Direction)
   END_RUNG
   RUNG wire#w2
      Move(in := 2, out1 => "Boxes".Boxes["Cnv2".Sect3.L.I_RFID_2].V_Direction)
   END_RUNG
   RUNG wire#w2
      P_Trig( "M_R1_Cont_Trig" )
      "Enqueue3"("Array" := "Cnv2".Sect3.L.V_ArrayOfBox, Input := "Cnv2".Sect3.L.I_RFID_2, size := "Cnv2".Sect3.L.V_NumOfBox)
   END_RUNG
   RUNG wire#w1
      Contact( "B_R1_Return" )
      wire#w3
      S_Coil( "M_B2L_S3_1" )
   END_RUNG
   RUNG wire#w3
      Move(in := 0, out1 => "Boxes".Boxes["Cnv2".Sect3.L.I_RFID_2].V_Destination[1], out2 => "Boxes".Boxes["Cnv2".Sect3.L.I_RFID_2].V_Destination[2], out3 => "Boxes".Boxes["Cnv2".Sect3.L.I_RFID_2].V_Destination[3], out4 => "Boxes".Boxes["Cnv2".Sect3.L.I_RFID_2].V_Completed["Boxes".Boxes["Cnv2".Sect3.L.I_RFID_2].V_NumOfComp])
   END_RUNG
   RUNG wire#w3
      Move(in := 2, out1 => "Cnv2".Sect3.Direction)
   END_RUNG
   RUNG wire#w3
      Move(in := 2, out1 => "Boxes".Boxes["Cnv2".Sect3.L.I_RFID_2].V_Direction)
   END_RUNG
   RUNG wire#w3
      P_Trig( "M_R1_Return_Trig" )
      "Enqueue3"("Array" := "Cnv2".Sect3.L.V_ArrayOfBox, Input := "Cnv2".Sect3.L.I_RFID_2, size := "Cnv2".Sect3.L.V_NumOfBox)
   END_RUNG
   // the same network as SCL:
   #_w1 := "M_R1_Start" AND "B_R1_Continue";
   IF #_w1 THEN
       "M_B2L_S3_1" := TRUE;
       "Cnv2".Sect3.Direction := 2;
       "Boxes".Boxes["Cnv2".Sect3.L.I_RFID_2].V_Direction := 2;
   END_IF;
   #_w2 := #_w1 AND NOT "M_R1_Cont_Trig";   // rising edge
   "M_R1_Cont_Trig" := #_w1;
   #_w3 := "M_R1_Start";
   IF #_w2 THEN
       "Enqueue3"("Array" := "Cnv2".Sect3.L.V_ArrayOfBox,
                  Input := "Cnv2".Sect3.L.I_RFID_2,
                  size := "Cnv2".Sect3.L.V_NumOfBox);
   END_IF;
   #_w4 := #_w3 AND "B_R1_Return";
   IF #_w4 THEN
       "M_B2L_S3_1" := TRUE;
       "Boxes".Boxes["Cnv2".Sect3.L.I_RFID_2].V_Destination[1] := 0;
       "Boxes".Boxes["Cnv2".Sect3.L.I_RFID_2].V_Destination[2] := 0;
       "Boxes".Boxes["Cnv2".Sect3.L.I_RFID_2].V_Destination[3] := 0;
       "Boxes".Boxes["Cnv2".Sect3.L.I_RFID_2].V_Completed["Boxes".Boxes["Cnv2".Sect3.L.I_RFID_2].V_NumOfComp] := 0;
       "Cnv2".Sect3.Direction := 2;
       "Boxes".Boxes["Cnv2".Sect3.L.I_RFID_2].V_Direction := 2;
   END_IF;
   #_w5 := #_w4 AND NOT "M_R1_Return_Trig";   // rising edge
   "M_R1_Return_Trig" := #_w4;
   IF #_w5 THEN
       "Enqueue3"("Array" := "Cnv2".Sect3.L.V_ArrayOfBox,
                  Input := "Cnv2".Sect3.L.I_RFID_2,
                  size := "Cnv2".Sect3.L.V_NumOfBox);
   END_IF;
END_REGION

REGION Network 92: Mode frw sect 4 high frw input - activate
   RUNG wire#powerrail
      Contact( "M_A_2to4_L1-L2_F4" )
      { S7_Templates := "SrcType := DInt" } GT_Contact(in1 := "Cnv2".Sect4.H.I_RFID_1, in2 := 0)
      { S7_Templates := "SrcType := Byte" } EQ_Contact(in1 := "Cnv2".Sect4.Direction, in2 := 1)
      S_Coil( "M_F2H_S4_1" )
   END_RUNG
   // the same network as SCL:
   IF "M_A_2to4_L1-L2_F4" AND ("Cnv2".Sect4.H.I_RFID_1 > 0) AND ("Cnv2".Sect4.Direction = 1) THEN
       "M_F2H_S4_1" := TRUE;
   END_IF;
END_REGION

REGION Network 93: Mode frw sect 4 high frw input
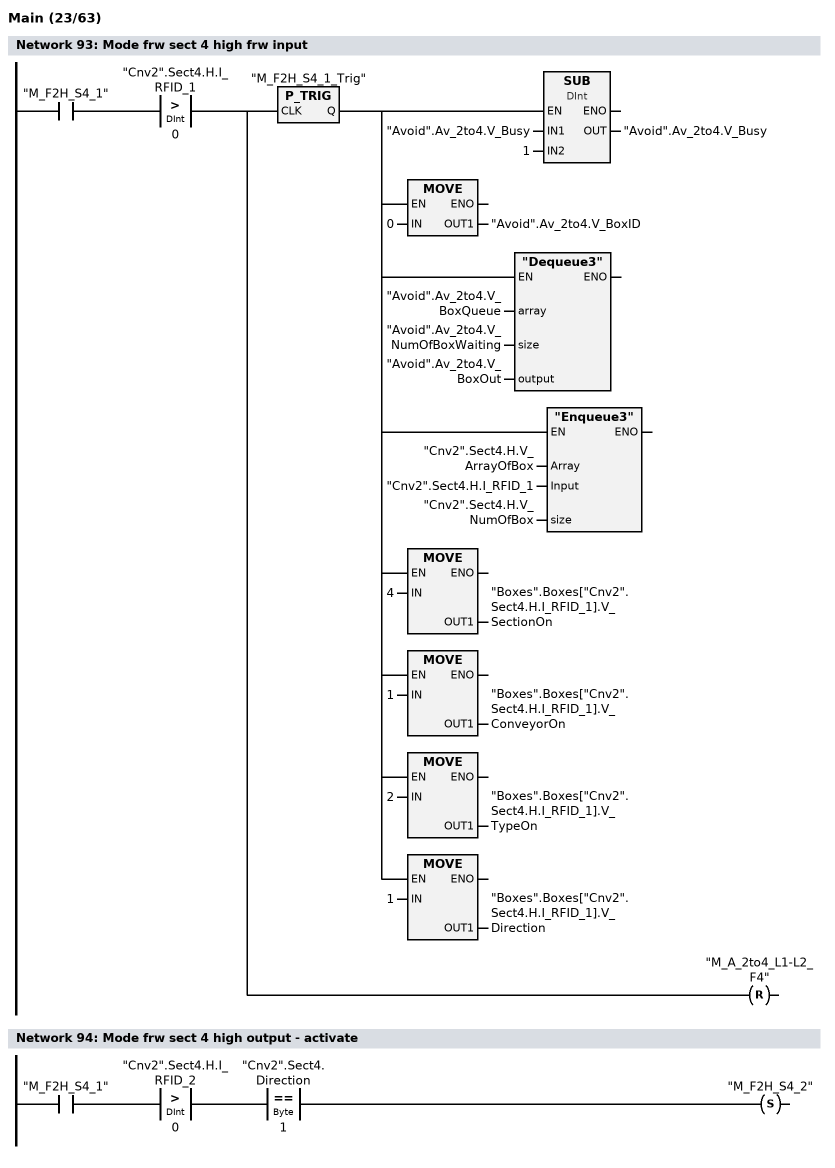
   RUNG wire#powerrail
      Contact( "M_F2H_S4_1" )
      { S7_Templates := "SrcType := DInt" } GT_Contact(in1 := "Cnv2".Sect4.H.I_RFID_1, in2 := 0)
      wire#w1
      P_Trig( "M_F2H_S4_1_Trig" )
      wire#w2
      { S7_Templates := "SrcType := DInt" } Sub(in1 := "Avoid".Av_2to4.V_Busy, in2 := 1, out => "Avoid".Av_2to4.V_Busy)
   END_RUNG
   RUNG wire#w2
      Move(in := 0, out1 => "Avoid".Av_2to4.V_BoxID)
   END_RUNG
   RUNG wire#w2
      "Dequeue3"("array" := "Avoid".Av_2to4.V_BoxQueue, size := "Avoid".Av_2to4.V_NumOfBoxWaiting, output := "Avoid".Av_2to4.V_BoxOut)
   END_RUNG
   RUNG wire#w2
      "Enqueue3"("Array" := "Cnv2".Sect4.H.V_ArrayOfBox, Input := "Cnv2".Sect4.H.I_RFID_1, size := "Cnv2".Sect4.H.V_NumOfBox)
   END_RUNG
   RUNG wire#w2
      Move(in := 4, out1 => "Boxes".Boxes["Cnv2".Sect4.H.I_RFID_1].V_SectionOn)
   END_RUNG
   RUNG wire#w2
      Move(in := 1, out1 => "Boxes".Boxes["Cnv2".Sect4.H.I_RFID_1].V_ConveyorOn)
   END_RUNG
   RUNG wire#w2
      Move(in := 2, out1 => "Boxes".Boxes["Cnv2".Sect4.H.I_RFID_1].V_TypeOn)
   END_RUNG
   RUNG wire#w2
      Move(in := 1, out1 => "Boxes".Boxes["Cnv2".Sect4.H.I_RFID_1].V_Direction)
   END_RUNG
   RUNG wire#w1
      R_Coil( "M_A_2to4_L1-L2_F4" )
   END_RUNG
   // the same network as SCL:
   #_w1 := "M_F2H_S4_1" AND ("Cnv2".Sect4.H.I_RFID_1 > 0);
   #_w2 := #_w1 AND NOT "M_F2H_S4_1_Trig";   // rising edge
   "M_F2H_S4_1_Trig" := #_w1;
   IF #_w2 THEN
       "Avoid".Av_2to4.V_Busy := "Avoid".Av_2to4.V_Busy - 1;
       "Avoid".Av_2to4.V_BoxID := 0;
       "Dequeue3"("array" := "Avoid".Av_2to4.V_BoxQueue,
                  size := "Avoid".Av_2to4.V_NumOfBoxWaiting,
                  output := "Avoid".Av_2to4.V_BoxOut);
       "Enqueue3"("Array" := "Cnv2".Sect4.H.V_ArrayOfBox,
                  Input := "Cnv2".Sect4.H.I_RFID_1,
                  size := "Cnv2".Sect4.H.V_NumOfBox);
       "Boxes".Boxes["Cnv2".Sect4.H.I_RFID_1].V_SectionOn := 4;
       "Boxes".Boxes["Cnv2".Sect4.H.I_RFID_1].V_ConveyorOn := 1;
       "Boxes".Boxes["Cnv2".Sect4.H.I_RFID_1].V_TypeOn := 2;
       "Boxes".Boxes["Cnv2".Sect4.H.I_RFID_1].V_Direction := 1;
   END_IF;
   IF #_w1 THEN "M_A_2to4_L1-L2_F4" := FALSE; END_IF;
END_REGION

REGION Network 94: Mode frw sect 4 high output - activate
   RUNG wire#powerrail
      Contact( "M_F2H_S4_1" )
      { S7_Templates := "SrcType := DInt" } GT_Contact(in1 := "Cnv2".Sect4.H.I_RFID_2, in2 := 0)
      { S7_Templates := "SrcType := Byte" } EQ_Contact(in1 := "Cnv2".Sect4.Direction, in2 := 1)
      S_Coil( "M_F2H_S4_2" )
   END_RUNG
   // the same network as SCL:
   IF "M_F2H_S4_1" AND ("Cnv2".Sect4.H.I_RFID_2 > 0) AND ("Cnv2".Sect4.Direction = 1) THEN
       "M_F2H_S4_2" := TRUE;
   END_IF;
END_REGION

REGION Network 95: Mode frw sect 4 high output
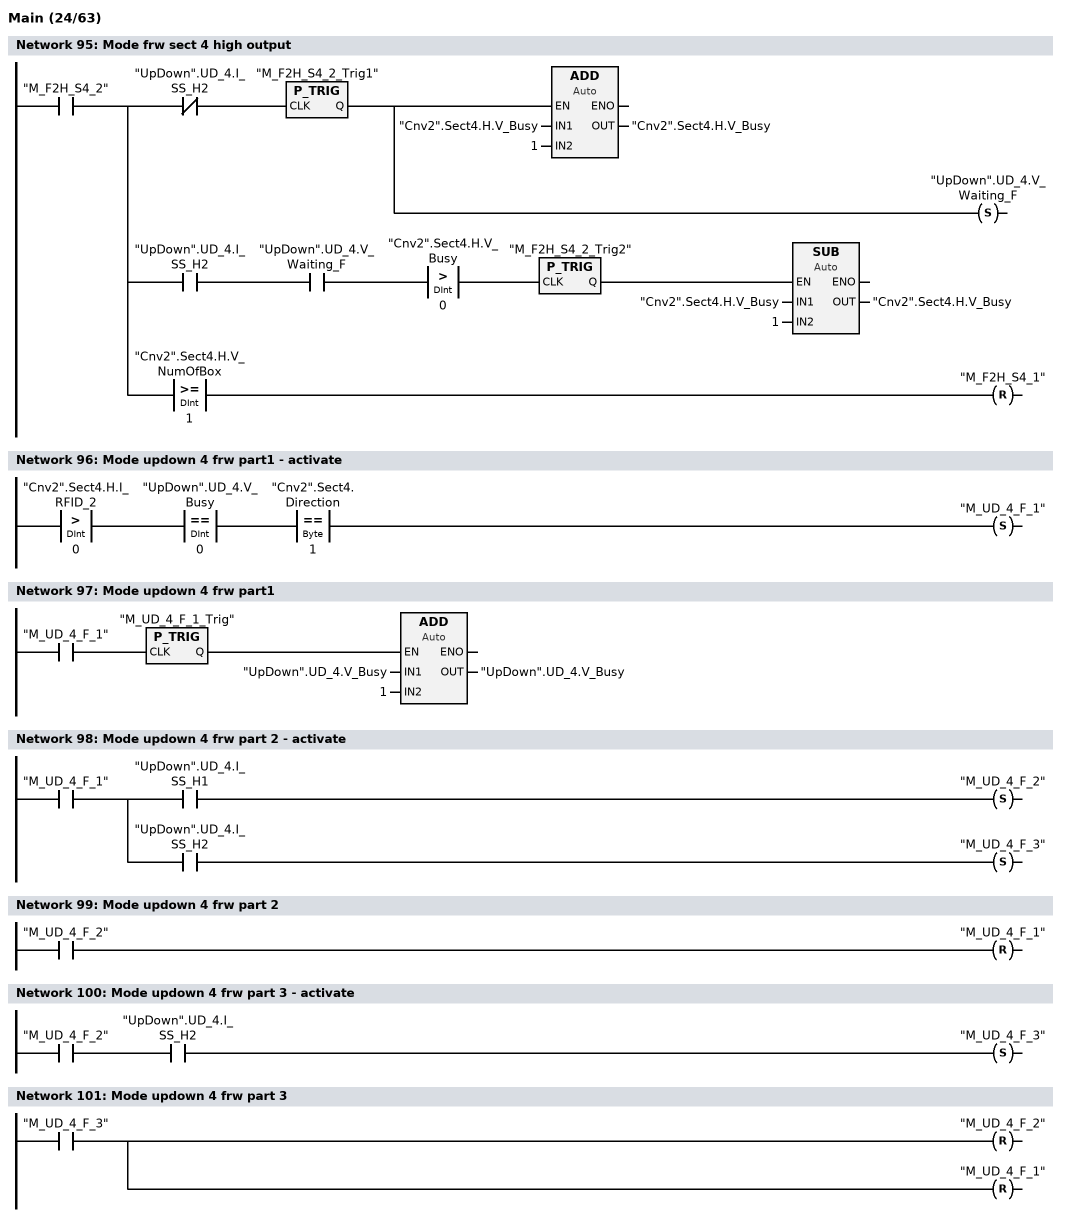
   RUNG wire#powerrail
      Contact( "M_F2H_S4_2" )
      wire#w1
      I_Contact( "UpDown".UD_4.I_SS_H2 )
      P_Trig( "M_F2H_S4_2_Trig1" )
      wire#w2
      Add(in1 := "Cnv2".Sect4.H.V_Busy, in2 := 1, out => "Cnv2".Sect4.H.V_Busy)
   END_RUNG
   RUNG wire#w2
      S_Coil( "UpDown".UD_4.V_Waiting_F )
   END_RUNG
   RUNG wire#w1
      Contact( "UpDown".UD_4.I_SS_H2 )
      Contact( "UpDown".UD_4.V_Waiting_F )
      { S7_Templates := "SrcType := DInt" } GT_Contact(in1 := "Cnv2".Sect4.H.V_Busy, in2 := 0)
      P_Trig( "M_F2H_S4_2_Trig2" )
      Sub(in1 := "Cnv2".Sect4.H.V_Busy, in2 := 1, out => "Cnv2".Sect4.H.V_Busy)
   END_RUNG
   RUNG wire#w1
      { S7_Templates := "SrcType := DInt" } GE_Contact(in1 := "Cnv2".Sect4.H.V_NumOfBox, in2 := 1)
      R_Coil( "M_F2H_S4_1" )
   END_RUNG
   // the same network as SCL:
   #_w1 := "M_F2H_S4_2" AND NOT "UpDown".UD_4.I_SS_H2;
   #_w2 := #_w1 AND NOT "M_F2H_S4_2_Trig1";   // rising edge
   "M_F2H_S4_2_Trig1" := #_w1;
   IF #_w2 THEN
       "Cnv2".Sect4.H.V_Busy := "Cnv2".Sect4.H.V_Busy + 1;
       "UpDown".UD_4.V_Waiting_F := TRUE;
   END_IF;
   #_w3 := "M_F2H_S4_2" AND "UpDown".UD_4.I_SS_H2 AND "UpDown".UD_4.V_Waiting_F AND ("Cnv2".Sect4.H.V_Busy > 0);
   #_w4 := #_w3 AND NOT "M_F2H_S4_2_Trig2";   // rising edge
   "M_F2H_S4_2_Trig2" := #_w3;
   IF #_w4 THEN "Cnv2".Sect4.H.V_Busy := "Cnv2".Sect4.H.V_Busy - 1; END_IF;
   IF "M_F2H_S4_2" AND ("Cnv2".Sect4.H.V_NumOfBox >= 1) THEN "M_F2H_S4_1" := FALSE; END_IF;
END_REGION

REGION Network 96: Mode updown 4 frw part1 - activate
   RUNG wire#powerrail
      { S7_Templates := "SrcType := DInt" } GT_Contact(in1 := "Cnv2".Sect4.H.I_RFID_2, in2 := 0)
      { S7_Templates := "SrcType := DInt" } EQ_Contact(in1 := "UpDown".UD_4.V_Busy, in2 := 0)
      { S7_Templates := "SrcType := Byte" } EQ_Contact(in1 := "Cnv2".Sect4.Direction, in2 := 1)
      S_Coil( "M_UD_4_F_1" )
   END_RUNG
   // the same network as SCL:
   IF ("Cnv2".Sect4.H.I_RFID_2 > 0) AND ("UpDown".UD_4.V_Busy = 0) AND ("Cnv2".Sect4.Direction = 1) THEN
       "M_UD_4_F_1" := TRUE;
   END_IF;
END_REGION

REGION Network 97: Mode updown 4 frw part1
   RUNG wire#powerrail
      Contact( "M_UD_4_F_1" )
      P_Trig( "M_UD_4_F_1_Trig" )
      Add(in1 := "UpDown".UD_4.V_Busy, in2 := 1, out => "UpDown".UD_4.V_Busy)
   END_RUNG
   // the same network as SCL:
   #_w1 := "M_UD_4_F_1" AND NOT "M_UD_4_F_1_Trig";   // rising edge
   "M_UD_4_F_1_Trig" := "M_UD_4_F_1";
   IF #_w1 THEN "UpDown".UD_4.V_Busy := "UpDown".UD_4.V_Busy + 1; END_IF;
END_REGION

REGION Network 98: Mode updown 4 frw part 2 - activate
   RUNG wire#powerrail
      Contact( "M_UD_4_F_1" )
      wire#w1
      Contact( "UpDown".UD_4.I_SS_H1 )
      S_Coil( "M_UD_4_F_2" )
   END_RUNG
   RUNG wire#w1
      Contact( "UpDown".UD_4.I_SS_H2 )
      S_Coil( "M_UD_4_F_3" )
   END_RUNG
   // the same network as SCL:
   IF "M_UD_4_F_1" AND "UpDown".UD_4.I_SS_H1 THEN "M_UD_4_F_2" := TRUE; END_IF;
   IF "M_UD_4_F_1" AND "UpDown".UD_4.I_SS_H2 THEN "M_UD_4_F_3" := TRUE; END_IF;
END_REGION

REGION Network 99: Mode updown 4 frw part 2
   RUNG wire#powerrail
      Contact( "M_UD_4_F_2" )
      R_Coil( "M_UD_4_F_1" )
   END_RUNG
   // the same network as SCL:
   IF "M_UD_4_F_2" THEN "M_UD_4_F_1" := FALSE; END_IF;
END_REGION

REGION Network 100: Mode updown 4 frw part 3 - activate
   RUNG wire#powerrail
      Contact( "M_UD_4_F_2" )
      Contact( "UpDown".UD_4.I_SS_H2 )
      S_Coil( "M_UD_4_F_3" )
   END_RUNG
   // the same network as SCL:
   IF "M_UD_4_F_2" AND "UpDown".UD_4.I_SS_H2 THEN "M_UD_4_F_3" := TRUE; END_IF;
END_REGION

REGION Network 101: Mode updown 4 frw part 3
   RUNG wire#powerrail
      Contact( "M_UD_4_F_3" )
      wire#w1
      R_Coil( "M_UD_4_F_2" )
   END_RUNG
   RUNG wire#w1
      R_Coil( "M_UD_4_F_1" )
   END_RUNG
   // the same network as SCL:
   IF "M_UD_4_F_3" THEN
       "M_UD_4_F_2" := FALSE;
       "M_UD_4_F_1" := FALSE;
   END_IF;
END_REGION

REGION Network 102: Mode updown 4 frw part 4 - activate
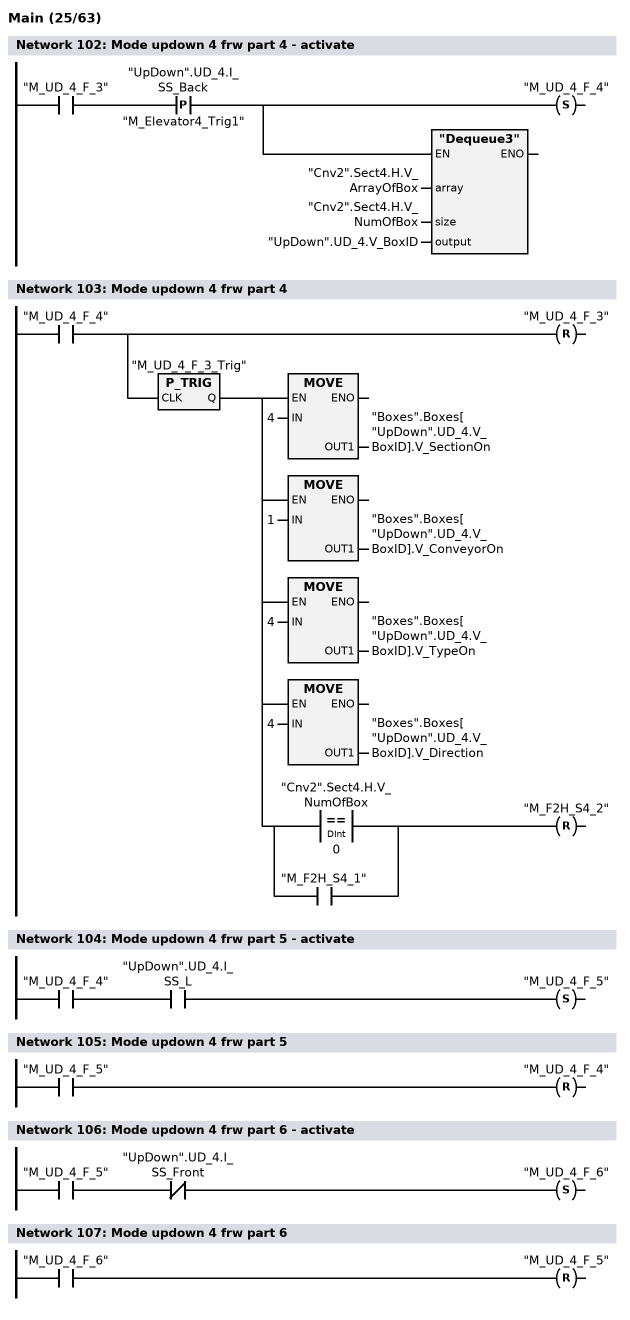
   RUNG wire#powerrail
      Contact( "M_UD_4_F_3" )
      P_Contact(operand := "UpDown".UD_4.I_SS_Back, bit := "M_Elevator4_Trig1")
      wire#w1
      S_Coil( "M_UD_4_F_4" )
   END_RUNG
   RUNG wire#w1
      "Dequeue3"("array" := "Cnv2".Sect4.H.V_ArrayOfBox, size := "Cnv2".Sect4.H.V_NumOfBox, output := "UpDown".UD_4.V_BoxID)
   END_RUNG
   // the same network as SCL:
   #_w1 := "M_UD_4_F_3" AND "UpDown".UD_4.I_SS_Back AND NOT "M_Elevator4_Trig1";   // rising edge of "UpDown".UD_4.I_SS_Back
   "M_Elevator4_Trig1" := "UpDown".UD_4.I_SS_Back;
   IF #_w1 THEN
       "M_UD_4_F_4" := TRUE;
       "Dequeue3"("array" := "Cnv2".Sect4.H.V_ArrayOfBox,
                  size := "Cnv2".Sect4.H.V_NumOfBox,
                  output := "UpDown".UD_4.V_BoxID);
   END_IF;
END_REGION

REGION Network 103: Mode updown 4 frw part 4
   RUNG wire#powerrail
      Contact( "M_UD_4_F_4" )
      wire#w1
      R_Coil( "M_UD_4_F_3" )
   END_RUNG
   RUNG wire#w1
      P_Trig( "M_UD_4_F_3_Trig" )
      wire#w2
      Move(in := 4, out1 => "Boxes".Boxes["UpDown".UD_4.V_BoxID].V_SectionOn)
   END_RUNG
   RUNG wire#w2
      Move(in := 1, out1 => "Boxes".Boxes["UpDown".UD_4.V_BoxID].V_ConveyorOn)
   END_RUNG
   RUNG wire#w2
      Move(in := 4, out1 => "Boxes".Boxes["UpDown".UD_4.V_BoxID].V_TypeOn)
   END_RUNG
   RUNG wire#w2
      Move(in := 4, out1 => "Boxes".Boxes["UpDown".UD_4.V_BoxID].V_Direction)
   END_RUNG
   RUNG wire#w2
      { S7_Templates := "SrcType := DInt" } EQ_Contact(in1 := "Cnv2".Sect4.H.V_NumOfBox, in2 := 0)
      wire#w3
      R_Coil( "M_F2H_S4_2" )
   END_RUNG
   RUNG wire#w2
      Contact( "M_F2H_S4_1" )
   END_RUNG wire#w3
   // the same network as SCL:
   IF "M_UD_4_F_4" THEN "M_UD_4_F_3" := FALSE; END_IF;
   #_w1 := "M_UD_4_F_4" AND NOT "M_UD_4_F_3_Trig";   // rising edge
   "M_UD_4_F_3_Trig" := "M_UD_4_F_4";
   IF #_w1 THEN
       "Boxes".Boxes["UpDown".UD_4.V_BoxID].V_SectionOn := 4;
       "Boxes".Boxes["UpDown".UD_4.V_BoxID].V_ConveyorOn := 1;
       "Boxes".Boxes["UpDown".UD_4.V_BoxID].V_TypeOn := 4;
       "Boxes".Boxes["UpDown".UD_4.V_BoxID].V_Direction := 4;
   END_IF;
   IF #_w1 AND (("Cnv2".Sect4.H.V_NumOfBox = 0) OR "M_F2H_S4_1") THEN "M_F2H_S4_2" := FALSE; END_IF;
END_REGION

REGION Network 104: Mode updown 4 frw part 5 - activate
   RUNG wire#powerrail
      Contact( "M_UD_4_F_4" )
      Contact( "UpDown".UD_4.I_SS_L )
      S_Coil( "M_UD_4_F_5" )
   END_RUNG
   // the same network as SCL:
   IF "M_UD_4_F_4" AND "UpDown".UD_4.I_SS_L THEN "M_UD_4_F_5" := TRUE; END_IF;
END_REGION

REGION Network 105: Mode updown 4 frw part 5
   RUNG wire#powerrail
      Contact( "M_UD_4_F_5" )
      R_Coil( "M_UD_4_F_4" )
   END_RUNG
   // the same network as SCL:
   IF "M_UD_4_F_5" THEN "M_UD_4_F_4" := FALSE; END_IF;
END_REGION

REGION Network 106: Mode updown 4 frw part 6 - activate
   RUNG wire#powerrail
      Contact( "M_UD_4_F_5" )
      I_Contact( "UpDown".UD_4.I_SS_Front )
      S_Coil( "M_UD_4_F_6" )
   END_RUNG
   // the same network as SCL:
   IF "M_UD_4_F_5" AND NOT "UpDown".UD_4.I_SS_Front THEN "M_UD_4_F_6" := TRUE; END_IF;
END_REGION

REGION Network 107: Mode updown 4 frw part 6
   RUNG wire#powerrail
      Contact( "M_UD_4_F_6" )
      R_Coil( "M_UD_4_F_5" )
   END_RUNG
   // the same network as SCL:
   IF "M_UD_4_F_6" THEN "M_UD_4_F_5" := FALSE; END_IF;
END_REGION

REGION Network 108: Mode updown 4 frw part 7 - activate
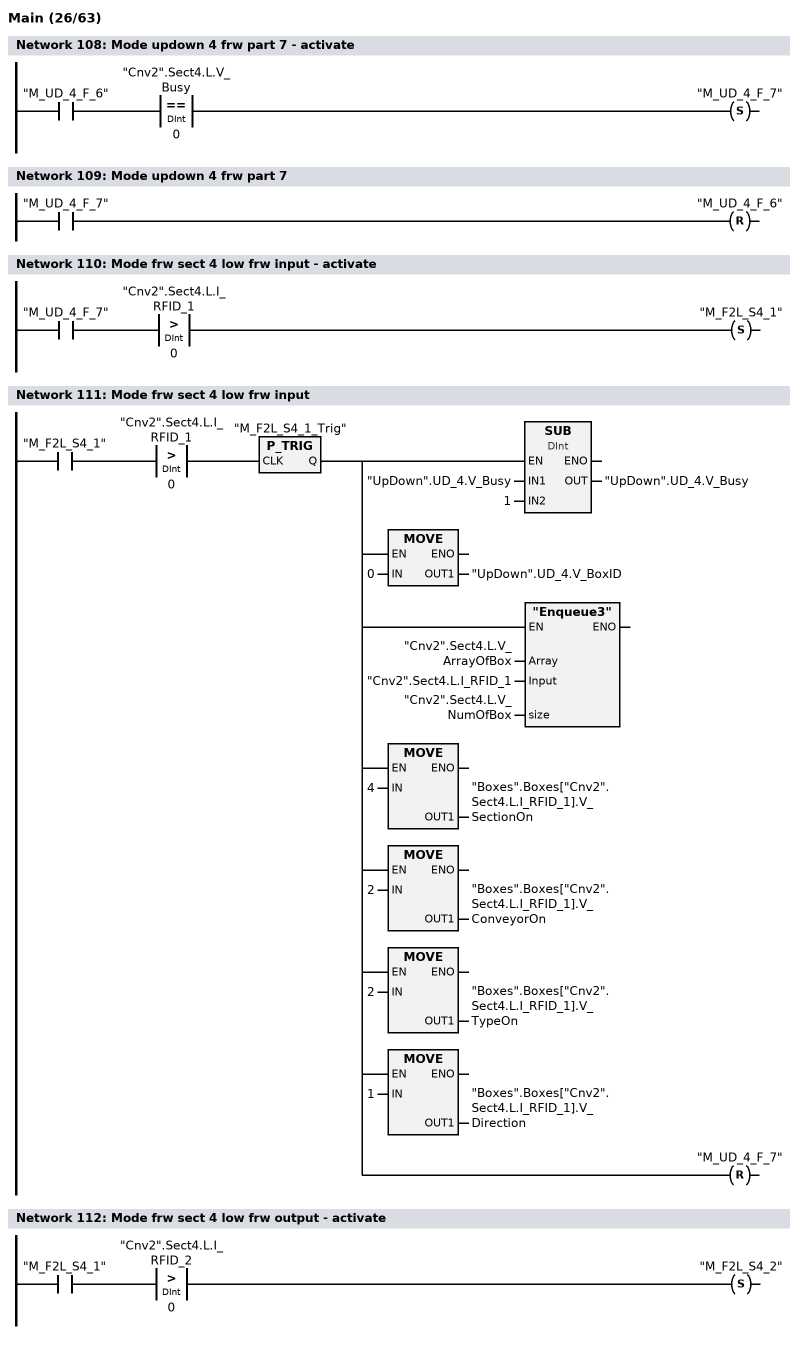
   RUNG wire#powerrail
      Contact( "M_UD_4_F_6" )
      { S7_Templates := "SrcType := DInt" } EQ_Contact(in1 := "Cnv2".Sect4.L.V_Busy, in2 := 0)
      S_Coil( "M_UD_4_F_7" )
   END_RUNG
   // the same network as SCL:
   IF "M_UD_4_F_6" AND ("Cnv2".Sect4.L.V_Busy = 0) THEN "M_UD_4_F_7" := TRUE; END_IF;
END_REGION

REGION Network 109: Mode updown 4 frw part 7
   RUNG wire#powerrail
      Contact( "M_UD_4_F_7" )
      R_Coil( "M_UD_4_F_6" )
   END_RUNG
   // the same network as SCL:
   IF "M_UD_4_F_7" THEN "M_UD_4_F_6" := FALSE; END_IF;
END_REGION

REGION Network 110: Mode frw sect 4 low frw input - activate
   RUNG wire#powerrail
      Contact( "M_UD_4_F_7" )
      { S7_Templates := "SrcType := DInt" } GT_Contact(in1 := "Cnv2".Sect4.L.I_RFID_1, in2 := 0)
      S_Coil( "M_F2L_S4_1" )
   END_RUNG
   // the same network as SCL:
   IF "M_UD_4_F_7" AND ("Cnv2".Sect4.L.I_RFID_1 > 0) THEN "M_F2L_S4_1" := TRUE; END_IF;
END_REGION

REGION Network 111: Mode frw sect 4 low frw input
   RUNG wire#powerrail
      Contact( "M_F2L_S4_1" )
      { S7_Templates := "SrcType := DInt" } GT_Contact(in1 := "Cnv2".Sect4.L.I_RFID_1, in2 := 0)
      P_Trig( "M_F2L_S4_1_Trig" )
      wire#w1
      { S7_Templates := "SrcType := DInt" } Sub(in1 := "UpDown".UD_4.V_Busy, in2 := 1, out => "UpDown".UD_4.V_Busy)
   END_RUNG
   RUNG wire#w1
      Move(in := 0, out1 => "UpDown".UD_4.V_BoxID)
   END_RUNG
   RUNG wire#w1
      "Enqueue3"("Array" := "Cnv2".Sect4.L.V_ArrayOfBox, Input := "Cnv2".Sect4.L.I_RFID_1, size := "Cnv2".Sect4.L.V_NumOfBox)
   END_RUNG
   RUNG wire#w1
      Move(in := 4, out1 => "Boxes".Boxes["Cnv2".Sect4.L.I_RFID_1].V_SectionOn)
   END_RUNG
   RUNG wire#w1
      Move(in := 2, out1 => "Boxes".Boxes["Cnv2".Sect4.L.I_RFID_1].V_ConveyorOn)
   END_RUNG
   RUNG wire#w1
      Move(in := 2, out1 => "Boxes".Boxes["Cnv2".Sect4.L.I_RFID_1].V_TypeOn)
   END_RUNG
   RUNG wire#w1
      Move(in := 1, out1 => "Boxes".Boxes["Cnv2".Sect4.L.I_RFID_1].V_Direction)
   END_RUNG
   RUNG wire#w1
      R_Coil( "M_UD_4_F_7" )
   END_RUNG
   // the same network as SCL:
   #_w1 := "M_F2L_S4_1" AND ("Cnv2".Sect4.L.I_RFID_1 > 0);
   #_w2 := #_w1 AND NOT "M_F2L_S4_1_Trig";   // rising edge
   "M_F2L_S4_1_Trig" := #_w1;
   IF #_w2 THEN
       "UpDown".UD_4.V_Busy := "UpDown".UD_4.V_Busy - 1;
       "UpDown".UD_4.V_BoxID := 0;
       "Enqueue3"("Array" := "Cnv2".Sect4.L.V_ArrayOfBox,
                  Input := "Cnv2".Sect4.L.I_RFID_1,
                  size := "Cnv2".Sect4.L.V_NumOfBox);
       "Boxes".Boxes["Cnv2".Sect4.L.I_RFID_1].V_SectionOn := 4;
       "Boxes".Boxes["Cnv2".Sect4.L.I_RFID_1].V_ConveyorOn := 2;
       "Boxes".Boxes["Cnv2".Sect4.L.I_RFID_1].V_TypeOn := 2;
       "Boxes".Boxes["Cnv2".Sect4.L.I_RFID_1].V_Direction := 1;
       "M_UD_4_F_7" := FALSE;
   END_IF;
END_REGION

REGION Network 112: Mode frw sect 4 low frw output - activate
   RUNG wire#powerrail
      Contact( "M_F2L_S4_1" )
      { S7_Templates := "SrcType := DInt" } GT_Contact(in1 := "Cnv2".Sect4.L.I_RFID_2, in2 := 0)
      S_Coil( "M_F2L_S4_2" )
   END_RUNG
   // the same network as SCL:
   IF "M_F2L_S4_1" AND ("Cnv2".Sect4.L.I_RFID_2 > 0) THEN "M_F2L_S4_2" := TRUE; END_IF;
END_REGION

REGION Network 113: Mode frw sect 4 low frw output
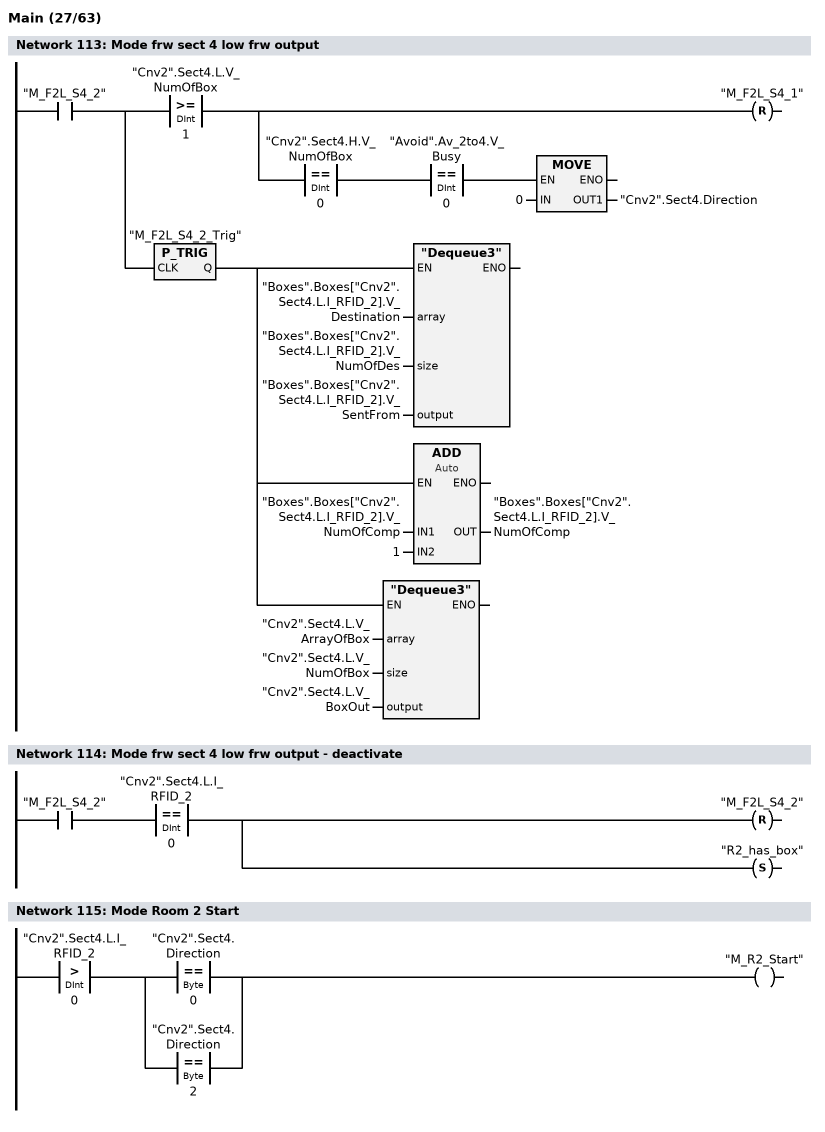
   RUNG wire#powerrail
      Contact( "M_F2L_S4_2" )
      wire#w1
      { S7_Templates := "SrcType := DInt" } GE_Contact(in1 := "Cnv2".Sect4.L.V_NumOfBox, in2 := 1)
      wire#w2
      R_Coil( "M_F2L_S4_1" )
   END_RUNG
   RUNG wire#w2
      { S7_Templates := "SrcType := DInt" } EQ_Contact(in1 := "Cnv2".Sect4.H.V_NumOfBox, in2 := 0)
      { S7_Templates := "SrcType := DInt" } EQ_Contact(in1 := "Avoid".Av_2to4.V_Busy, in2 := 0)
      Move(in := 0, out1 => "Cnv2".Sect4.Direction)
   END_RUNG
   RUNG wire#w1
      P_Trig( "M_F2L_S4_2_Trig" )
      wire#w3
      "Dequeue3"("array" := "Boxes".Boxes["Cnv2".Sect4.L.I_RFID_2].V_Destination, size := "Boxes".Boxes["Cnv2".Sect4.L.I_RFID_2].V_NumOfDes, output := "Boxes".Boxes["Cnv2".Sect4.L.I_RFID_2].V_SentFrom)
   END_RUNG
   RUNG wire#w3
      Add(in1 := "Boxes".Boxes["Cnv2".Sect4.L.I_RFID_2].V_NumOfComp, in2 := 1, out => "Boxes".Boxes["Cnv2".Sect4.L.I_RFID_2].V_NumOfComp)
   END_RUNG
   RUNG wire#w3
      "Dequeue3"("array" := "Cnv2".Sect4.L.V_ArrayOfBox, size := "Cnv2".Sect4.L.V_NumOfBox, output := "Cnv2".Sect4.L.V_BoxOut)
   END_RUNG
   // the same network as SCL:
   #_w1 := "M_F2L_S4_2" AND ("Cnv2".Sect4.L.V_NumOfBox >= 1);
   IF #_w1 THEN "M_F2L_S4_1" := FALSE; END_IF;
   IF #_w1 AND ("Cnv2".Sect4.H.V_NumOfBox = 0) AND ("Avoid".Av_2to4.V_Busy = 0) THEN
       "Cnv2".Sect4.Direction := 0;
   END_IF;
   #_w2 := "M_F2L_S4_2" AND NOT "M_F2L_S4_2_Trig";   // rising edge
   "M_F2L_S4_2_Trig" := "M_F2L_S4_2";
   IF #_w2 THEN
       "Dequeue3"("array" := "Boxes".Boxes["Cnv2".Sect4.L.I_RFID_2].V_Destination,
                  size := "Boxes".Boxes["Cnv2".Sect4.L.I_RFID_2].V_NumOfDes,
                  output := "Boxes".Boxes["Cnv2".Sect4.L.I_RFID_2].V_SentFrom);
       "Boxes".Boxes["Cnv2".Sect4.L.I_RFID_2].V_NumOfComp := "Boxes".Boxes["Cnv2".Sect4.L.I_RFID_2].V_NumOfComp + 1;
       "Dequeue3"("array" := "Cnv2".Sect4.L.V_ArrayOfBox,
                  size := "Cnv2".Sect4.L.V_NumOfBox,
                  output := "Cnv2".Sect4.L.V_BoxOut);
   END_IF;
END_REGION

REGION Network 114: Mode frw sect 4 low frw output - deactivate
   RUNG wire#powerrail
      Contact( "M_F2L_S4_2" )
      { S7_Templates := "SrcType := DInt" } EQ_Contact(in1 := "Cnv2".Sect4.L.I_RFID_2, in2 := 0)
      wire#w1
      R_Coil( "M_F2L_S4_2" )
   END_RUNG
   RUNG wire#w1
      S_Coil( "R2_has_box" )
   END_RUNG
   // the same network as SCL:
   #_w1 := "M_F2L_S4_2" AND ("Cnv2".Sect4.L.I_RFID_2 = 0);
   IF #_w1 THEN
       "M_F2L_S4_2" := FALSE;
       "R2_has_box" := TRUE;
   END_IF;
END_REGION

REGION Network 115: Mode Room 2 Start
   RUNG wire#powerrail
      { S7_Templates := "SrcType := DInt" } GT_Contact(in1 := "Cnv2".Sect4.L.I_RFID_2, in2 := 0)
      wire#w1
      { S7_Templates := "SrcType := Byte" } EQ_Contact(in1 := "Cnv2".Sect4.Direction, in2 := 0)
      wire#w2
      Coil( "M_R2_Start" )
   END_RUNG
   RUNG wire#w1
      { S7_Templates := "SrcType := Byte" } EQ_Contact(in1 := "Cnv2".Sect4.Direction, in2 := 2)
   END_RUNG wire#w2
   // the same network as SCL:
   "M_R2_Start" := ("Cnv2".Sect4.L.I_RFID_2 > 0) AND (("Cnv2".Sect4.Direction = 0) OR ("Cnv2".Sect4.Direction = 2));
END_REGION

REGION Network 116: Mode Room 2 - choose return or continue and Mode back sect 3 input - activate
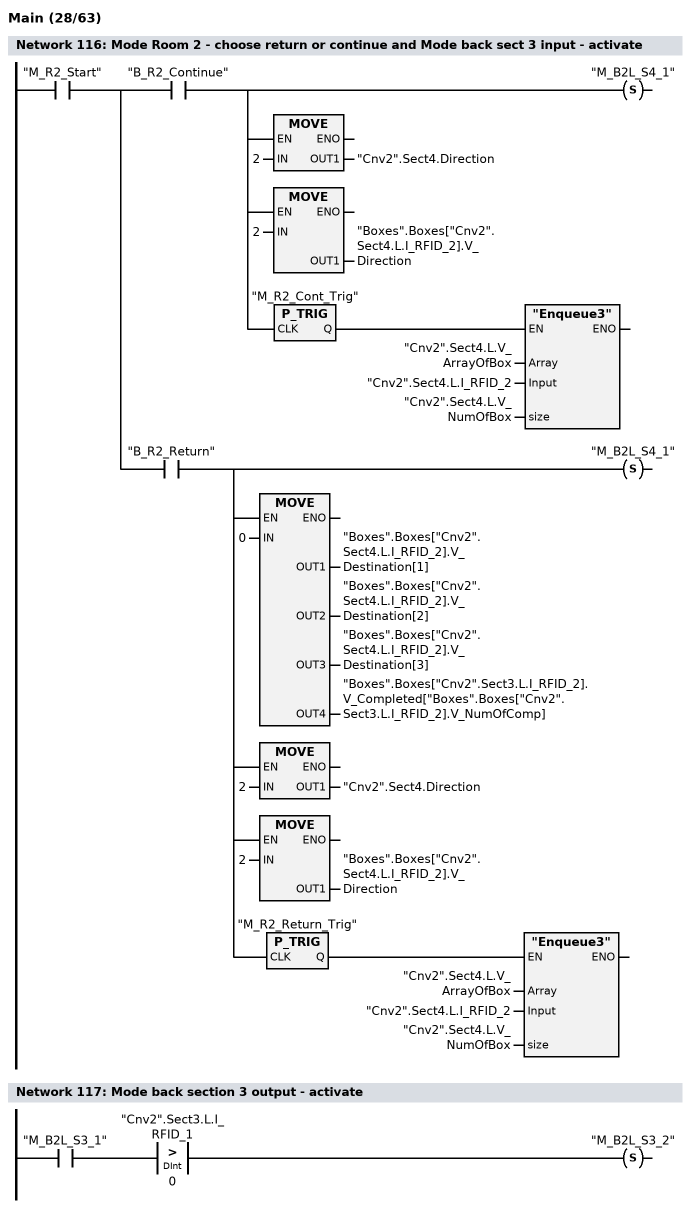
   RUNG wire#powerrail
      Contact( "M_R2_Start" )
      wire#w1
      Contact( "B_R2_Continue" )
      wire#w2
      S_Coil( "M_B2L_S4_1" )
   END_RUNG
   RUNG wire#w2
      Move(in := 2, out1 => "Cnv2".Sect4.Direction)
   END_RUNG
   RUNG wire#w2
      Move(in := 2, out1 => "Boxes".Boxes["Cnv2".Sect4.L.I_RFID_2].V_Direction)
   END_RUNG
   RUNG wire#w2
      P_Trig( "M_R2_Cont_Trig" )
      "Enqueue3"("Array" := "Cnv2".Sect4.L.V_ArrayOfBox, Input := "Cnv2".Sect4.L.I_RFID_2, size := "Cnv2".Sect4.L.V_NumOfBox)
   END_RUNG
   RUNG wire#w1
      Contact( "B_R2_Return" )
      wire#w3
      S_Coil( "M_B2L_S4_1" )
   END_RUNG
   RUNG wire#w3
      Move(in := 0, out1 => "Boxes".Boxes["Cnv2".Sect4.L.I_RFID_2].V_Destination[1], out2 => "Boxes".Boxes["Cnv2".Sect4.L.I_RFID_2].V_Destination[2], out3 => "Boxes".Boxes["Cnv2".Sect4.L.I_RFID_2].V_Destination[3], out4 => "Boxes".Boxes["Cnv2".Sect3.L.I_RFID_2].V_Completed["Boxes".Boxes["Cnv2".Sect3.L.I_RFID_2].V_NumOfComp])
   END_RUNG
   RUNG wire#w3
      Move(in := 2, out1 => "Cnv2".Sect4.Direction)
   END_RUNG
   RUNG wire#w3
      Move(in := 2, out1 => "Boxes".Boxes["Cnv2".Sect4.L.I_RFID_2].V_Direction)
   END_RUNG
   RUNG wire#w3
      P_Trig( "M_R2_Return_Trig" )
      "Enqueue3"("Array" := "Cnv2".Sect4.L.V_ArrayOfBox, Input := "Cnv2".Sect4.L.I_RFID_2, size := "Cnv2".Sect4.L.V_NumOfBox)
   END_RUNG
   // the same network as SCL:
   #_w1 := "M_R2_Start" AND "B_R2_Continue";
   IF #_w1 THEN
       "M_B2L_S4_1" := TRUE;
       "Cnv2".Sect4.Direction := 2;
       "Boxes".Boxes["Cnv2".Sect4.L.I_RFID_2].V_Direction := 2;
   END_IF;
   #_w2 := #_w1 AND NOT "M_R2_Cont_Trig";   // rising edge
   "M_R2_Cont_Trig" := #_w1;
   #_w3 := "M_R2_Start";
   IF #_w2 THEN
       "Enqueue3"("Array" := "Cnv2".Sect4.L.V_ArrayOfBox,
                  Input := "Cnv2".Sect4.L.I_RFID_2,
                  size := "Cnv2".Sect4.L.V_NumOfBox);
   END_IF;
   #_w4 := #_w3 AND "B_R2_Return";
   IF #_w4 THEN
       "M_B2L_S4_1" := TRUE;
       "Boxes".Boxes["Cnv2".Sect4.L.I_RFID_2].V_Destination[1] := 0;
       "Boxes".Boxes["Cnv2".Sect4.L.I_RFID_2].V_Destination[2] := 0;
       "Boxes".Boxes["Cnv2".Sect4.L.I_RFID_2].V_Destination[3] := 0;
       "Boxes".Boxes["Cnv2".Sect3.L.I_RFID_2].V_Completed["Boxes".Boxes["Cnv2".Sect3.L.I_RFID_2].V_NumOfComp] := 0;
       "Cnv2".Sect4.Direction := 2;
       "Boxes".Boxes["Cnv2".Sect4.L.I_RFID_2].V_Direction := 2;
   END_IF;
   #_w5 := #_w4 AND NOT "M_R2_Return_Trig";   // rising edge
   "M_R2_Return_Trig" := #_w4;
   IF #_w5 THEN
       "Enqueue3"("Array" := "Cnv2".Sect4.L.V_ArrayOfBox,
                  Input := "Cnv2".Sect4.L.I_RFID_2,
                  size := "Cnv2".Sect4.L.V_NumOfBox);
   END_IF;
END_REGION

REGION Network 117: Mode back section 3 output - activate
   RUNG wire#powerrail
      Contact( "M_B2L_S3_1" )
      { S7_Templates := "SrcType := DInt" } GT_Contact(in1 := "Cnv2".Sect3.L.I_RFID_1, in2 := 0)
      S_Coil( "M_B2L_S3_2" )
   END_RUNG
   // the same network as SCL:
   IF "M_B2L_S3_1" AND ("Cnv2".Sect3.L.I_RFID_1 > 0) THEN "M_B2L_S3_2" := TRUE; END_IF;
END_REGION

REGION Network 118: Mode back section 3 output
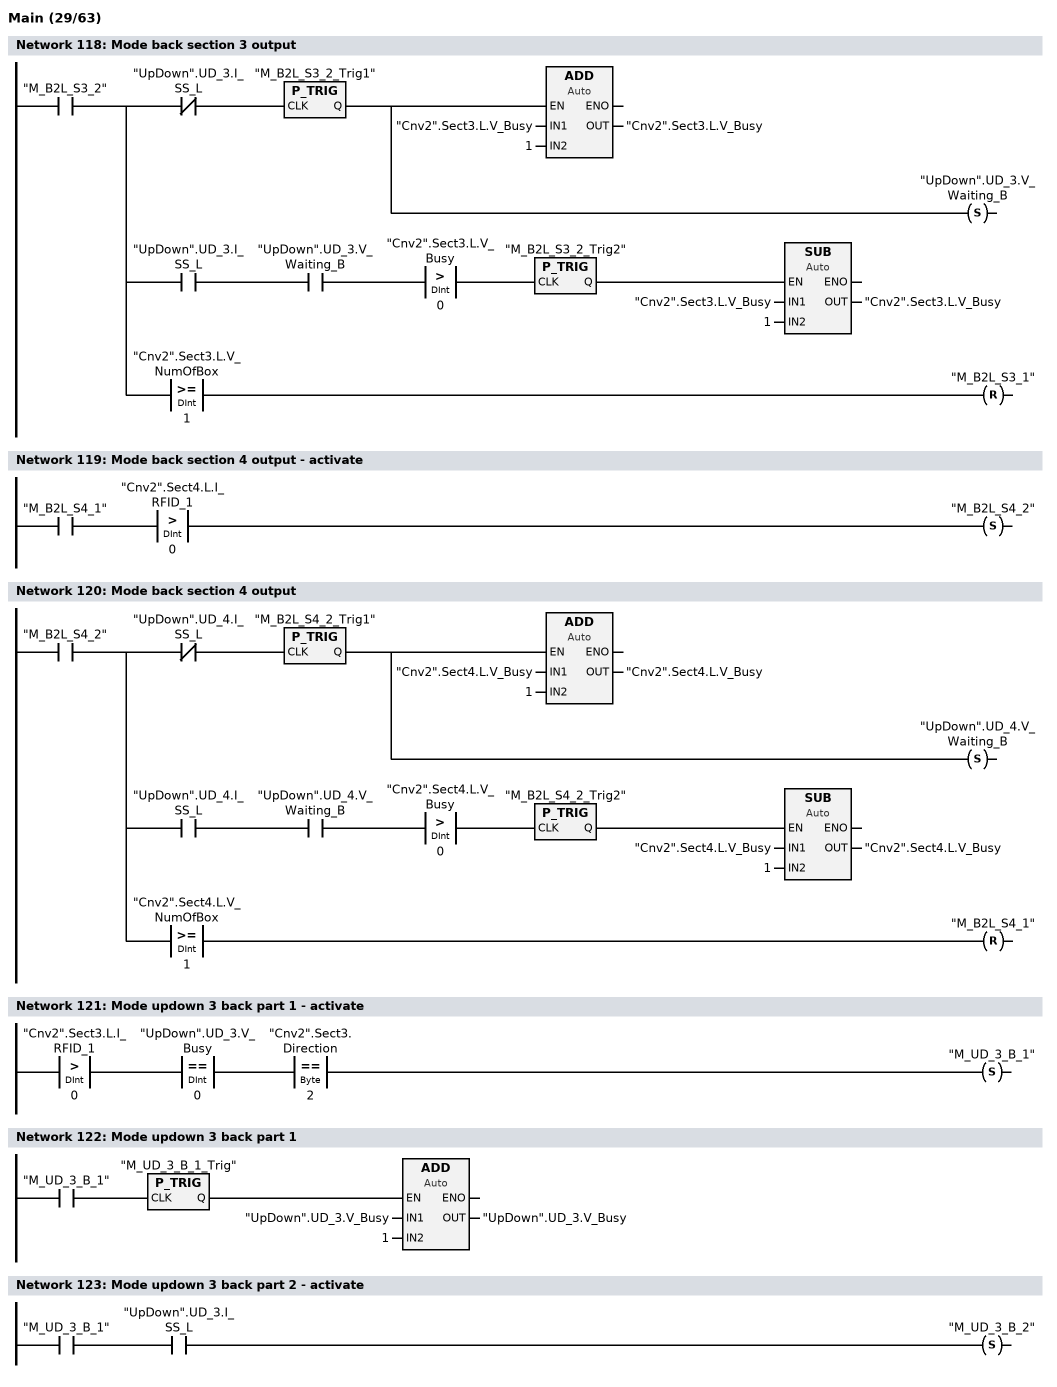
   RUNG wire#powerrail
      Contact( "M_B2L_S3_2" )
      wire#w1
      I_Contact( "UpDown".UD_3.I_SS_L )
      P_Trig( "M_B2L_S3_2_Trig1" )
      wire#w2
      Add(in1 := "Cnv2".Sect3.L.V_Busy, in2 := 1, out => "Cnv2".Sect3.L.V_Busy)
   END_RUNG
   RUNG wire#w2
      S_Coil( "UpDown".UD_3.V_Waiting_B )
   END_RUNG
   RUNG wire#w1
      Contact( "UpDown".UD_3.I_SS_L )
      Contact( "UpDown".UD_3.V_Waiting_B )
      { S7_Templates := "SrcType := DInt" } GT_Contact(in1 := "Cnv2".Sect3.L.V_Busy, in2 := 0)
      P_Trig( "M_B2L_S3_2_Trig2" )
      Sub(in1 := "Cnv2".Sect3.L.V_Busy, in2 := 1, out => "Cnv2".Sect3.L.V_Busy)
   END_RUNG
   RUNG wire#w1
      { S7_Templates := "SrcType := DInt" } GE_Contact(in1 := "Cnv2".Sect3.L.V_NumOfBox, in2 := 1)
      R_Coil( "M_B2L_S3_1" )
   END_RUNG
   // the same network as SCL:
   #_w1 := "M_B2L_S3_2" AND NOT "UpDown".UD_3.I_SS_L;
   #_w2 := #_w1 AND NOT "M_B2L_S3_2_Trig1";   // rising edge
   "M_B2L_S3_2_Trig1" := #_w1;
   IF #_w2 THEN
       "Cnv2".Sect3.L.V_Busy := "Cnv2".Sect3.L.V_Busy + 1;
       "UpDown".UD_3.V_Waiting_B := TRUE;
   END_IF;
   #_w3 := "M_B2L_S3_2" AND "UpDown".UD_3.I_SS_L AND "UpDown".UD_3.V_Waiting_B AND ("Cnv2".Sect3.L.V_Busy > 0);
   #_w4 := #_w3 AND NOT "M_B2L_S3_2_Trig2";   // rising edge
   "M_B2L_S3_2_Trig2" := #_w3;
   IF #_w4 THEN "Cnv2".Sect3.L.V_Busy := "Cnv2".Sect3.L.V_Busy - 1; END_IF;
   IF "M_B2L_S3_2" AND ("Cnv2".Sect3.L.V_NumOfBox >= 1) THEN "M_B2L_S3_1" := FALSE; END_IF;
END_REGION

REGION Network 119: Mode back section 4 output - activate
   RUNG wire#powerrail
      Contact( "M_B2L_S4_1" )
      { S7_Templates := "SrcType := DInt" } GT_Contact(in1 := "Cnv2".Sect4.L.I_RFID_1, in2 := 0)
      S_Coil( "M_B2L_S4_2" )
   END_RUNG
   // the same network as SCL:
   IF "M_B2L_S4_1" AND ("Cnv2".Sect4.L.I_RFID_1 > 0) THEN "M_B2L_S4_2" := TRUE; END_IF;
END_REGION

REGION Network 120: Mode back section 4 output
   RUNG wire#powerrail
      Contact( "M_B2L_S4_2" )
      wire#w1
      I_Contact( "UpDown".UD_4.I_SS_L )
      P_Trig( "M_B2L_S4_2_Trig1" )
      wire#w2
      Add(in1 := "Cnv2".Sect4.L.V_Busy, in2 := 1, out => "Cnv2".Sect4.L.V_Busy)
   END_RUNG
   RUNG wire#w2
      S_Coil( "UpDown".UD_4.V_Waiting_B )
   END_RUNG
   RUNG wire#w1
      Contact( "UpDown".UD_4.I_SS_L )
      Contact( "UpDown".UD_4.V_Waiting_B )
      { S7_Templates := "SrcType := DInt" } GT_Contact(in1 := "Cnv2".Sect4.L.V_Busy, in2 := 0)
      P_Trig( "M_B2L_S4_2_Trig2" )
      Sub(in1 := "Cnv2".Sect4.L.V_Busy, in2 := 1, out => "Cnv2".Sect4.L.V_Busy)
   END_RUNG
   RUNG wire#w1
      { S7_Templates := "SrcType := DInt" } GE_Contact(in1 := "Cnv2".Sect4.L.V_NumOfBox, in2 := 1)
      R_Coil( "M_B2L_S4_1" )
   END_RUNG
   // the same network as SCL:
   #_w1 := "M_B2L_S4_2" AND NOT "UpDown".UD_4.I_SS_L;
   #_w2 := #_w1 AND NOT "M_B2L_S4_2_Trig1";   // rising edge
   "M_B2L_S4_2_Trig1" := #_w1;
   IF #_w2 THEN
       "Cnv2".Sect4.L.V_Busy := "Cnv2".Sect4.L.V_Busy + 1;
       "UpDown".UD_4.V_Waiting_B := TRUE;
   END_IF;
   #_w3 := "M_B2L_S4_2" AND "UpDown".UD_4.I_SS_L AND "UpDown".UD_4.V_Waiting_B AND ("Cnv2".Sect4.L.V_Busy > 0);
   #_w4 := #_w3 AND NOT "M_B2L_S4_2_Trig2";   // rising edge
   "M_B2L_S4_2_Trig2" := #_w3;
   IF #_w4 THEN "Cnv2".Sect4.L.V_Busy := "Cnv2".Sect4.L.V_Busy - 1; END_IF;
   IF "M_B2L_S4_2" AND ("Cnv2".Sect4.L.V_NumOfBox >= 1) THEN "M_B2L_S4_1" := FALSE; END_IF;
END_REGION

REGION Network 121: Mode updown 3 back part 1 - activate
   RUNG wire#powerrail
      { S7_Templates := "SrcType := DInt" } GT_Contact(in1 := "Cnv2".Sect3.L.I_RFID_1, in2 := 0)
      { S7_Templates := "SrcType := DInt" } EQ_Contact(in1 := "UpDown".UD_3.V_Busy, in2 := 0)
      { S7_Templates := "SrcType := Byte" } EQ_Contact(in1 := "Cnv2".Sect3.Direction, in2 := 2)
      S_Coil( "M_UD_3_B_1" )
   END_RUNG
   // the same network as SCL:
   IF ("Cnv2".Sect3.L.I_RFID_1 > 0) AND ("UpDown".UD_3.V_Busy = 0) AND ("Cnv2".Sect3.Direction = 2) THEN
       "M_UD_3_B_1" := TRUE;
   END_IF;
END_REGION

REGION Network 122: Mode updown 3 back part 1
   RUNG wire#powerrail
      Contact( "M_UD_3_B_1" )
      P_Trig( "M_UD_3_B_1_Trig" )
      Add(in1 := "UpDown".UD_3.V_Busy, in2 := 1, out => "UpDown".UD_3.V_Busy)
   END_RUNG
   // the same network as SCL:
   #_w1 := "M_UD_3_B_1" AND NOT "M_UD_3_B_1_Trig";   // rising edge
   "M_UD_3_B_1_Trig" := "M_UD_3_B_1";
   IF #_w1 THEN "UpDown".UD_3.V_Busy := "UpDown".UD_3.V_Busy + 1; END_IF;
END_REGION

REGION Network 123: Mode updown 3 back part 2 - activate
   RUNG wire#powerrail
      Contact( "M_UD_3_B_1" )
      Contact( "UpDown".UD_3.I_SS_L )
      S_Coil( "M_UD_3_B_2" )
   END_RUNG
   // the same network as SCL:
   IF "M_UD_3_B_1" AND "UpDown".UD_3.I_SS_L THEN "M_UD_3_B_2" := TRUE; END_IF;
END_REGION

REGION Network 124: Mode updown 3 back part 2
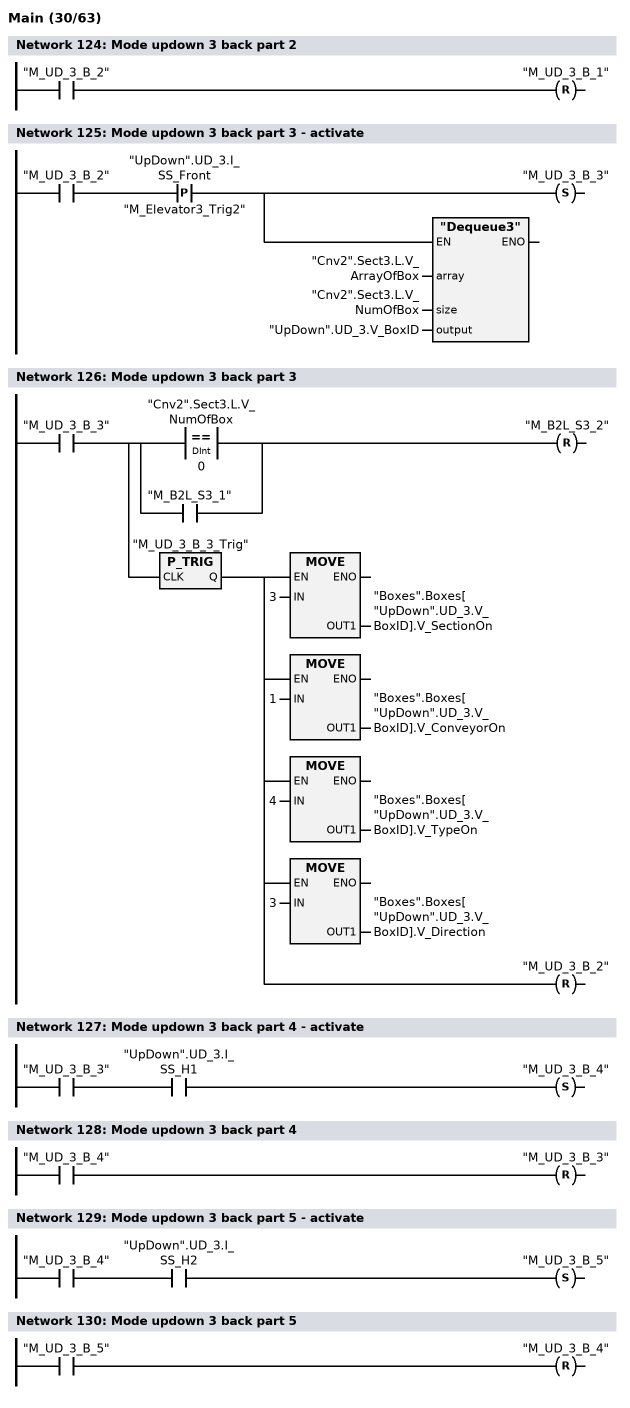
   RUNG wire#powerrail
      Contact( "M_UD_3_B_2" )
      R_Coil( "M_UD_3_B_1" )
   END_RUNG
   // the same network as SCL:
   IF "M_UD_3_B_2" THEN "M_UD_3_B_1" := FALSE; END_IF;
END_REGION

REGION Network 125: Mode updown 3 back part 3 - activate
   RUNG wire#powerrail
      Contact( "M_UD_3_B_2" )
      P_Contact(operand := "UpDown".UD_3.I_SS_Front, bit := "M_Elevator3_Trig2")
      wire#w1
      S_Coil( "M_UD_3_B_3" )
   END_RUNG
   RUNG wire#w1
      "Dequeue3"("array" := "Cnv2".Sect3.L.V_ArrayOfBox, size := "Cnv2".Sect3.L.V_NumOfBox, output := "UpDown".UD_3.V_BoxID)
   END_RUNG
   // the same network as SCL:
   #_w1 := "M_UD_3_B_2" AND "UpDown".UD_3.I_SS_Front AND NOT "M_Elevator3_Trig2";   // rising edge of "UpDown".UD_3.I_SS_Front
   "M_Elevator3_Trig2" := "UpDown".UD_3.I_SS_Front;
   IF #_w1 THEN
       "M_UD_3_B_3" := TRUE;
       "Dequeue3"("array" := "Cnv2".Sect3.L.V_ArrayOfBox,
                  size := "Cnv2".Sect3.L.V_NumOfBox,
                  output := "UpDown".UD_3.V_BoxID);
   END_IF;
END_REGION

REGION Network 126: Mode updown 3 back part 3
   RUNG wire#powerrail
      Contact( "M_UD_3_B_3" )
      wire#w1
      { S7_Templates := "SrcType := DInt" } EQ_Contact(in1 := "Cnv2".Sect3.L.V_NumOfBox, in2 := 0)
      wire#w2
      R_Coil( "M_B2L_S3_2" )
   END_RUNG
   RUNG wire#w1
      Contact( "M_B2L_S3_1" )
   END_RUNG wire#w2
   RUNG wire#w1
      P_Trig( "M_UD_3_B_3_Trig" )
      wire#w3
      Move(in := 3, out1 => "Boxes".Boxes["UpDown".UD_3.V_BoxID].V_SectionOn)
   END_RUNG
   RUNG wire#w3
      Move(in := 1, out1 => "Boxes".Boxes["UpDown".UD_3.V_BoxID].V_ConveyorOn)
   END_RUNG
   RUNG wire#w3
      Move(in := 4, out1 => "Boxes".Boxes["UpDown".UD_3.V_BoxID].V_TypeOn)
   END_RUNG
   RUNG wire#w3
      Move(in := 3, out1 => "Boxes".Boxes["UpDown".UD_3.V_BoxID].V_Direction)
   END_RUNG
   RUNG wire#w3
      R_Coil( "M_UD_3_B_2" )
   END_RUNG
   // the same network as SCL:
   IF "M_UD_3_B_3" AND (("Cnv2".Sect3.L.V_NumOfBox = 0) OR "M_B2L_S3_1") THEN "M_B2L_S3_2" := FALSE; END_IF;
   #_w1 := "M_UD_3_B_3" AND NOT "M_UD_3_B_3_Trig";   // rising edge
   "M_UD_3_B_3_Trig" := "M_UD_3_B_3";
   IF #_w1 THEN
       "Boxes".Boxes["UpDown".UD_3.V_BoxID].V_SectionOn := 3;
       "Boxes".Boxes["UpDown".UD_3.V_BoxID].V_ConveyorOn := 1;
       "Boxes".Boxes["UpDown".UD_3.V_BoxID].V_TypeOn := 4;
       "Boxes".Boxes["UpDown".UD_3.V_BoxID].V_Direction := 3;
       "M_UD_3_B_2" := FALSE;
   END_IF;
END_REGION

REGION Network 127: Mode updown 3 back part 4 - activate
   RUNG wire#powerrail
      Contact( "M_UD_3_B_3" )
      Contact( "UpDown".UD_3.I_SS_H1 )
      S_Coil( "M_UD_3_B_4" )
   END_RUNG
   // the same network as SCL:
   IF "M_UD_3_B_3" AND "UpDown".UD_3.I_SS_H1 THEN "M_UD_3_B_4" := TRUE; END_IF;
END_REGION

REGION Network 128: Mode updown 3 back part 4
   RUNG wire#powerrail
      Contact( "M_UD_3_B_4" )
      R_Coil( "M_UD_3_B_3" )
   END_RUNG
   // the same network as SCL:
   IF "M_UD_3_B_4" THEN "M_UD_3_B_3" := FALSE; END_IF;
END_REGION

REGION Network 129: Mode updown 3 back part 5 - activate
   RUNG wire#powerrail
      Contact( "M_UD_3_B_4" )
      Contact( "UpDown".UD_3.I_SS_H2 )
      S_Coil( "M_UD_3_B_5" )
   END_RUNG
   // the same network as SCL:
   IF "M_UD_3_B_4" AND "UpDown".UD_3.I_SS_H2 THEN "M_UD_3_B_5" := TRUE; END_IF;
END_REGION

REGION Network 130: Mode updown 3 back part 5
   RUNG wire#powerrail
      Contact( "M_UD_3_B_5" )
      R_Coil( "M_UD_3_B_4" )
   END_RUNG
   // the same network as SCL:
   IF "M_UD_3_B_5" THEN "M_UD_3_B_4" := FALSE; END_IF;
END_REGION

REGION Network 131: Mode updown 3 back part 6 - activate
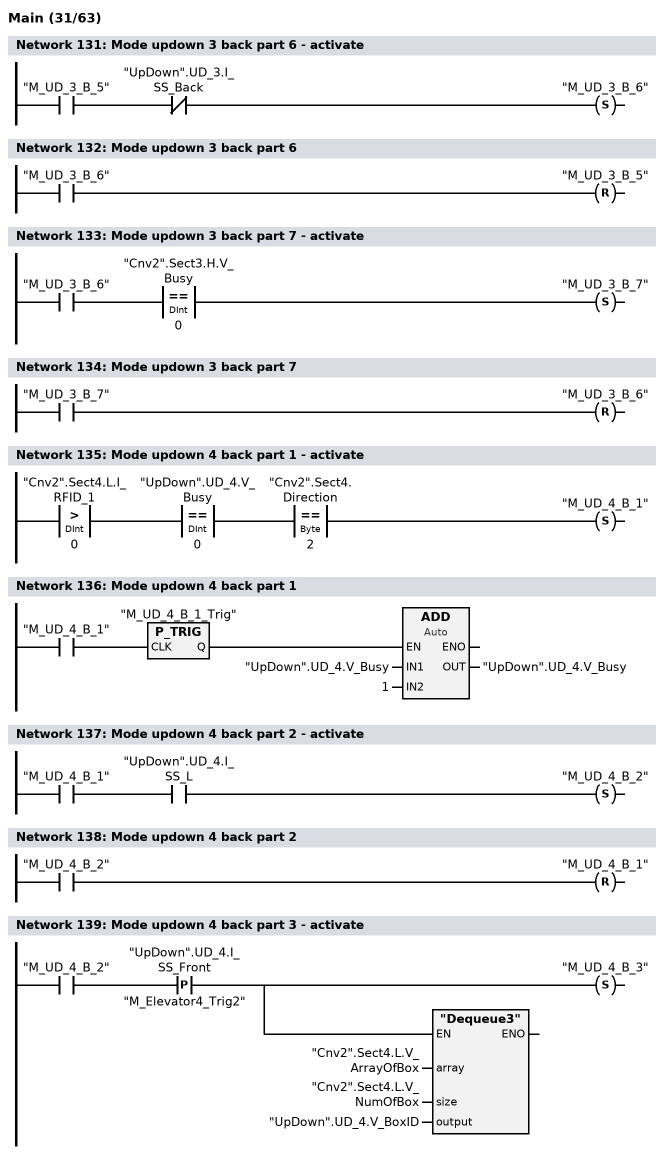
   RUNG wire#powerrail
      Contact( "M_UD_3_B_5" )
      I_Contact( "UpDown".UD_3.I_SS_Back )
      S_Coil( "M_UD_3_B_6" )
   END_RUNG
   // the same network as SCL:
   IF "M_UD_3_B_5" AND NOT "UpDown".UD_3.I_SS_Back THEN "M_UD_3_B_6" := TRUE; END_IF;
END_REGION

REGION Network 132: Mode updown 3 back part 6
   RUNG wire#powerrail
      Contact( "M_UD_3_B_6" )
      R_Coil( "M_UD_3_B_5" )
   END_RUNG
   // the same network as SCL:
   IF "M_UD_3_B_6" THEN "M_UD_3_B_5" := FALSE; END_IF;
END_REGION

REGION Network 133: Mode updown 3 back part 7 - activate
   RUNG wire#powerrail
      Contact( "M_UD_3_B_6" )
      { S7_Templates := "SrcType := DInt" } EQ_Contact(in1 := "Cnv2".Sect3.H.V_Busy, in2 := 0)
      S_Coil( "M_UD_3_B_7" )
   END_RUNG
   // the same network as SCL:
   IF "M_UD_3_B_6" AND ("Cnv2".Sect3.H.V_Busy = 0) THEN "M_UD_3_B_7" := TRUE; END_IF;
END_REGION

REGION Network 134: Mode updown 3 back part 7
   RUNG wire#powerrail
      Contact( "M_UD_3_B_7" )
      R_Coil( "M_UD_3_B_6" )
   END_RUNG
   // the same network as SCL:
   IF "M_UD_3_B_7" THEN "M_UD_3_B_6" := FALSE; END_IF;
END_REGION

REGION Network 135: Mode updown 4 back part 1 - activate
   RUNG wire#powerrail
      { S7_Templates := "SrcType := DInt" } GT_Contact(in1 := "Cnv2".Sect4.L.I_RFID_1, in2 := 0)
      { S7_Templates := "SrcType := DInt" } EQ_Contact(in1 := "UpDown".UD_4.V_Busy, in2 := 0)
      { S7_Templates := "SrcType := Byte" } EQ_Contact(in1 := "Cnv2".Sect4.Direction, in2 := 2)
      S_Coil( "M_UD_4_B_1" )
   END_RUNG
   // the same network as SCL:
   IF ("Cnv2".Sect4.L.I_RFID_1 > 0) AND ("UpDown".UD_4.V_Busy = 0) AND ("Cnv2".Sect4.Direction = 2) THEN
       "M_UD_4_B_1" := TRUE;
   END_IF;
END_REGION

REGION Network 136: Mode updown 4 back part 1
   RUNG wire#powerrail
      Contact( "M_UD_4_B_1" )
      P_Trig( "M_UD_4_B_1_Trig" )
      Add(in1 := "UpDown".UD_4.V_Busy, in2 := 1, out => "UpDown".UD_4.V_Busy)
   END_RUNG
   // the same network as SCL:
   #_w1 := "M_UD_4_B_1" AND NOT "M_UD_4_B_1_Trig";   // rising edge
   "M_UD_4_B_1_Trig" := "M_UD_4_B_1";
   IF #_w1 THEN "UpDown".UD_4.V_Busy := "UpDown".UD_4.V_Busy + 1; END_IF;
END_REGION

REGION Network 137: Mode updown 4 back part 2 - activate
   RUNG wire#powerrail
      Contact( "M_UD_4_B_1" )
      Contact( "UpDown".UD_4.I_SS_L )
      S_Coil( "M_UD_4_B_2" )
   END_RUNG
   // the same network as SCL:
   IF "M_UD_4_B_1" AND "UpDown".UD_4.I_SS_L THEN "M_UD_4_B_2" := TRUE; END_IF;
END_REGION

REGION Network 138: Mode updown 4 back part 2
   RUNG wire#powerrail
      Contact( "M_UD_4_B_2" )
      R_Coil( "M_UD_4_B_1" )
   END_RUNG
   // the same network as SCL:
   IF "M_UD_4_B_2" THEN "M_UD_4_B_1" := FALSE; END_IF;
END_REGION

REGION Network 139: Mode updown 4 back part 3 - activate
   RUNG wire#powerrail
      Contact( "M_UD_4_B_2" )
      P_Contact(operand := "UpDown".UD_4.I_SS_Front, bit := "M_Elevator4_Trig2")
      wire#w1
      S_Coil( "M_UD_4_B_3" )
   END_RUNG
   RUNG wire#w1
      "Dequeue3"("array" := "Cnv2".Sect4.L.V_ArrayOfBox, size := "Cnv2".Sect4.L.V_NumOfBox, output := "UpDown".UD_4.V_BoxID)
   END_RUNG
   // the same network as SCL:
   #_w1 := "M_UD_4_B_2" AND "UpDown".UD_4.I_SS_Front AND NOT "M_Elevator4_Trig2";   // rising edge of "UpDown".UD_4.I_SS_Front
   "M_Elevator4_Trig2" := "UpDown".UD_4.I_SS_Front;
   IF #_w1 THEN
       "M_UD_4_B_3" := TRUE;
       "Dequeue3"("array" := "Cnv2".Sect4.L.V_ArrayOfBox,
                  size := "Cnv2".Sect4.L.V_NumOfBox,
                  output := "UpDown".UD_4.V_BoxID);
   END_IF;
END_REGION

REGION Network 140: Mode updown 4 back part 3
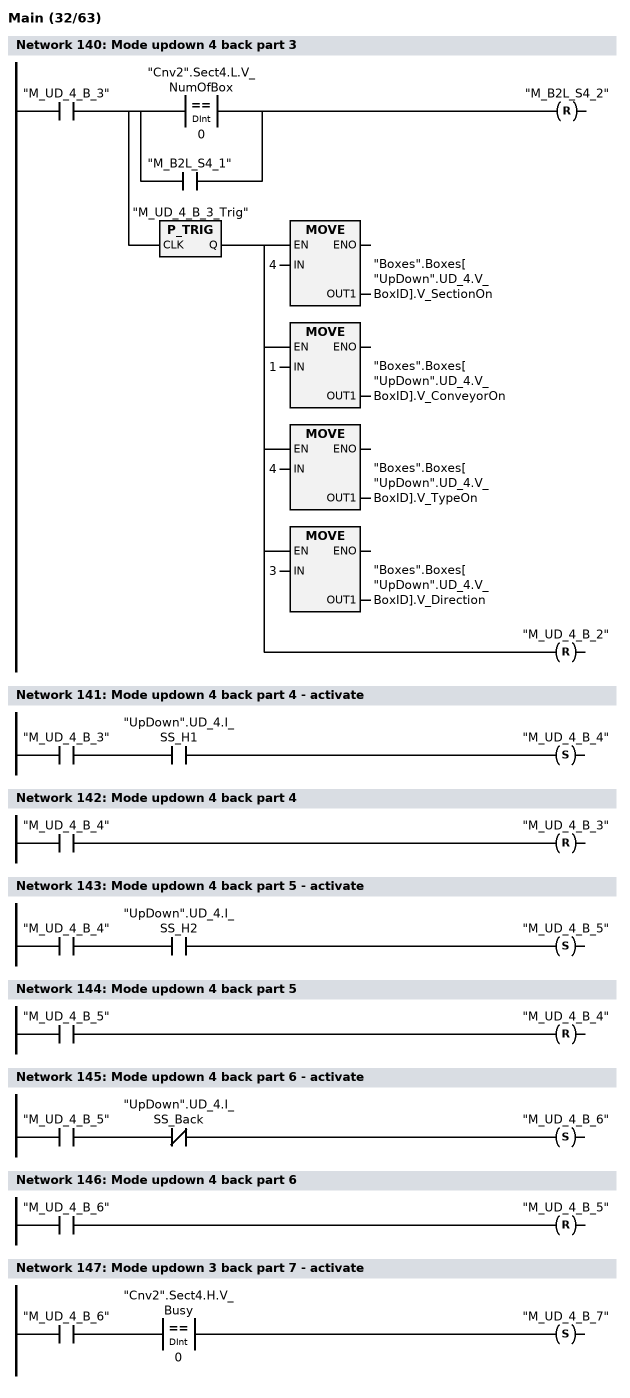
   RUNG wire#powerrail
      Contact( "M_UD_4_B_3" )
      wire#w1
      { S7_Templates := "SrcType := DInt" } EQ_Contact(in1 := "Cnv2".Sect4.L.V_NumOfBox, in2 := 0)
      wire#w2
      R_Coil( "M_B2L_S4_2" )
   END_RUNG
   RUNG wire#w1
      Contact( "M_B2L_S4_1" )
   END_RUNG wire#w2
   RUNG wire#w1
      P_Trig( "M_UD_4_B_3_Trig" )
      wire#w3
      Move(in := 4, out1 => "Boxes".Boxes["UpDown".UD_4.V_BoxID].V_SectionOn)
   END_RUNG
   RUNG wire#w3
      Move(in := 1, out1 => "Boxes".Boxes["UpDown".UD_4.V_BoxID].V_ConveyorOn)
   END_RUNG
   RUNG wire#w3
      Move(in := 4, out1 => "Boxes".Boxes["UpDown".UD_4.V_BoxID].V_TypeOn)
   END_RUNG
   RUNG wire#w3
      Move(in := 3, out1 => "Boxes".Boxes["UpDown".UD_4.V_BoxID].V_Direction)
   END_RUNG
   RUNG wire#w3
      R_Coil( "M_UD_4_B_2" )
   END_RUNG
   // the same network as SCL:
   IF "M_UD_4_B_3" AND (("Cnv2".Sect4.L.V_NumOfBox = 0) OR "M_B2L_S4_1") THEN "M_B2L_S4_2" := FALSE; END_IF;
   #_w1 := "M_UD_4_B_3" AND NOT "M_UD_4_B_3_Trig";   // rising edge
   "M_UD_4_B_3_Trig" := "M_UD_4_B_3";
   IF #_w1 THEN
       "Boxes".Boxes["UpDown".UD_4.V_BoxID].V_SectionOn := 4;
       "Boxes".Boxes["UpDown".UD_4.V_BoxID].V_ConveyorOn := 1;
       "Boxes".Boxes["UpDown".UD_4.V_BoxID].V_TypeOn := 4;
       "Boxes".Boxes["UpDown".UD_4.V_BoxID].V_Direction := 3;
       "M_UD_4_B_2" := FALSE;
   END_IF;
END_REGION

REGION Network 141: Mode updown 4 back part 4 - activate
   RUNG wire#powerrail
      Contact( "M_UD_4_B_3" )
      Contact( "UpDown".UD_4.I_SS_H1 )
      S_Coil( "M_UD_4_B_4" )
   END_RUNG
   // the same network as SCL:
   IF "M_UD_4_B_3" AND "UpDown".UD_4.I_SS_H1 THEN "M_UD_4_B_4" := TRUE; END_IF;
END_REGION

REGION Network 142: Mode updown 4 back part 4
   RUNG wire#powerrail
      Contact( "M_UD_4_B_4" )
      R_Coil( "M_UD_4_B_3" )
   END_RUNG
   // the same network as SCL:
   IF "M_UD_4_B_4" THEN "M_UD_4_B_3" := FALSE; END_IF;
END_REGION

REGION Network 143: Mode updown 4 back part 5 - activate
   RUNG wire#powerrail
      Contact( "M_UD_4_B_4" )
      Contact( "UpDown".UD_4.I_SS_H2 )
      S_Coil( "M_UD_4_B_5" )
   END_RUNG
   // the same network as SCL:
   IF "M_UD_4_B_4" AND "UpDown".UD_4.I_SS_H2 THEN "M_UD_4_B_5" := TRUE; END_IF;
END_REGION

REGION Network 144: Mode updown 4 back part 5
   RUNG wire#powerrail
      Contact( "M_UD_4_B_5" )
      R_Coil( "M_UD_4_B_4" )
   END_RUNG
   // the same network as SCL:
   IF "M_UD_4_B_5" THEN "M_UD_4_B_4" := FALSE; END_IF;
END_REGION

REGION Network 145: Mode updown 4 back part 6 - activate
   RUNG wire#powerrail
      Contact( "M_UD_4_B_5" )
      I_Contact( "UpDown".UD_4.I_SS_Back )
      S_Coil( "M_UD_4_B_6" )
   END_RUNG
   // the same network as SCL:
   IF "M_UD_4_B_5" AND NOT "UpDown".UD_4.I_SS_Back THEN "M_UD_4_B_6" := TRUE; END_IF;
END_REGION

REGION Network 146: Mode updown 4 back part 6
   RUNG wire#powerrail
      Contact( "M_UD_4_B_6" )
      R_Coil( "M_UD_4_B_5" )
   END_RUNG
   // the same network as SCL:
   IF "M_UD_4_B_6" THEN "M_UD_4_B_5" := FALSE; END_IF;
END_REGION

REGION Network 147: Mode updown 3 back part 7 - activate
   RUNG wire#powerrail
      Contact( "M_UD_4_B_6" )
      { S7_Templates := "SrcType := DInt" } EQ_Contact(in1 := "Cnv2".Sect4.H.V_Busy, in2 := 0)
      S_Coil( "M_UD_4_B_7" )
   END_RUNG
   // the same network as SCL:
   IF "M_UD_4_B_6" AND ("Cnv2".Sect4.H.V_Busy = 0) THEN "M_UD_4_B_7" := TRUE; END_IF;
END_REGION

REGION Network 148: Mode updown 3 back part 7
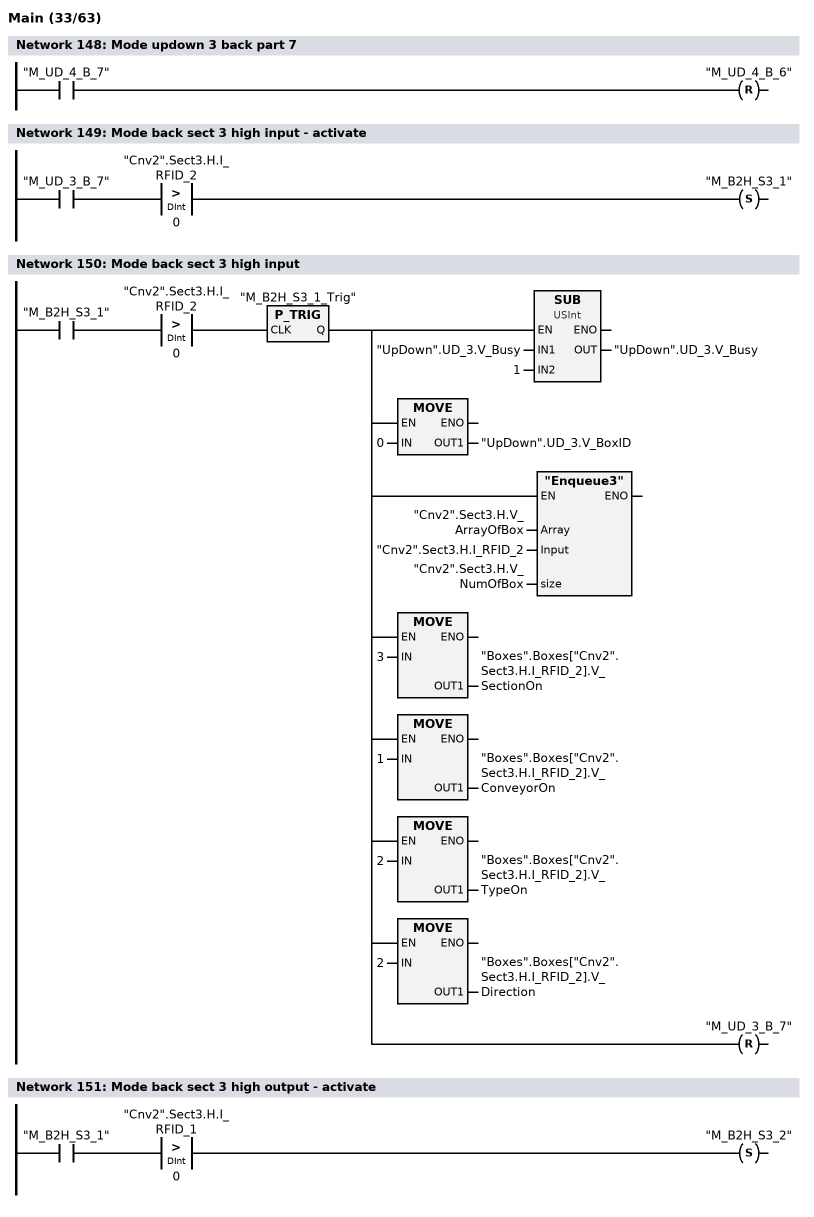
   RUNG wire#powerrail
      Contact( "M_UD_4_B_7" )
      R_Coil( "M_UD_4_B_6" )
   END_RUNG
   // the same network as SCL:
   IF "M_UD_4_B_7" THEN "M_UD_4_B_6" := FALSE; END_IF;
END_REGION

REGION Network 149: Mode back sect 3 high input - activate
   RUNG wire#powerrail
      Contact( "M_UD_3_B_7" )
      { S7_Templates := "SrcType := DInt" } GT_Contact(in1 := "Cnv2".Sect3.H.I_RFID_2, in2 := 0)
      S_Coil( "M_B2H_S3_1" )
   END_RUNG
   // the same network as SCL:
   IF "M_UD_3_B_7" AND ("Cnv2".Sect3.H.I_RFID_2 > 0) THEN "M_B2H_S3_1" := TRUE; END_IF;
END_REGION

REGION Network 150: Mode back sect 3 high input
   RUNG wire#powerrail
      Contact( "M_B2H_S3_1" )
      { S7_Templates := "SrcType := DInt" } GT_Contact(in1 := "Cnv2".Sect3.H.I_RFID_2, in2 := 0)
      P_Trig( "M_B2H_S3_1_Trig" )
      wire#w1
      { S7_Templates := "SrcType := USInt" } Sub(in1 := "UpDown".UD_3.V_Busy, in2 := 1, out => "UpDown".UD_3.V_Busy)
   END_RUNG
   RUNG wire#w1
      Move(in := 0, out1 => "UpDown".UD_3.V_BoxID)
   END_RUNG
   RUNG wire#w1
      "Enqueue3"("Array" := "Cnv2".Sect3.H.V_ArrayOfBox, Input := "Cnv2".Sect3.H.I_RFID_2, size := "Cnv2".Sect3.H.V_NumOfBox)
   END_RUNG
   RUNG wire#w1
      Move(in := 3, out1 => "Boxes".Boxes["Cnv2".Sect3.H.I_RFID_2].V_SectionOn)
   END_RUNG
   RUNG wire#w1
      Move(in := 1, out1 => "Boxes".Boxes["Cnv2".Sect3.H.I_RFID_2].V_ConveyorOn)
   END_RUNG
   RUNG wire#w1
      Move(in := 2, out1 => "Boxes".Boxes["Cnv2".Sect3.H.I_RFID_2].V_TypeOn)
   END_RUNG
   RUNG wire#w1
      Move(in := 2, out1 => "Boxes".Boxes["Cnv2".Sect3.H.I_RFID_2].V_Direction)
   END_RUNG
   RUNG wire#w1
      R_Coil( "M_UD_3_B_7" )
   END_RUNG
   // the same network as SCL:
   #_w1 := "M_B2H_S3_1" AND ("Cnv2".Sect3.H.I_RFID_2 > 0);
   #_w2 := #_w1 AND NOT "M_B2H_S3_1_Trig";   // rising edge
   "M_B2H_S3_1_Trig" := #_w1;
   IF #_w2 THEN
       "UpDown".UD_3.V_Busy := "UpDown".UD_3.V_Busy - 1;
       "UpDown".UD_3.V_BoxID := 0;
       "Enqueue3"("Array" := "Cnv2".Sect3.H.V_ArrayOfBox,
                  Input := "Cnv2".Sect3.H.I_RFID_2,
                  size := "Cnv2".Sect3.H.V_NumOfBox);
       "Boxes".Boxes["Cnv2".Sect3.H.I_RFID_2].V_SectionOn := 3;
       "Boxes".Boxes["Cnv2".Sect3.H.I_RFID_2].V_ConveyorOn := 1;
       "Boxes".Boxes["Cnv2".Sect3.H.I_RFID_2].V_TypeOn := 2;
       "Boxes".Boxes["Cnv2".Sect3.H.I_RFID_2].V_Direction := 2;
       "M_UD_3_B_7" := FALSE;
   END_IF;
END_REGION

REGION Network 151: Mode back sect 3 high output - activate
   RUNG wire#powerrail
      Contact( "M_B2H_S3_1" )
      { S7_Templates := "SrcType := DInt" } GT_Contact(in1 := "Cnv2".Sect3.H.I_RFID_1, in2 := 0)
      S_Coil( "M_B2H_S3_2" )
   END_RUNG
   // the same network as SCL:
   IF "M_B2H_S3_1" AND ("Cnv2".Sect3.H.I_RFID_1 > 0) THEN "M_B2H_S3_2" := TRUE; END_IF;
END_REGION

REGION Network 152: Mode back sect 3 high output
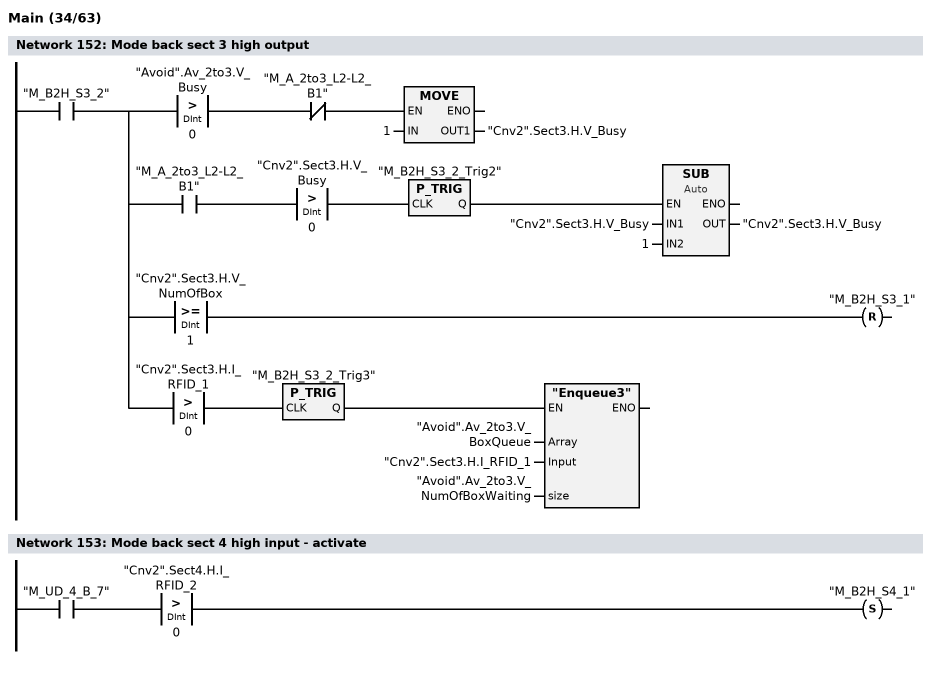
   RUNG wire#powerrail
      Contact( "M_B2H_S3_2" )
      wire#w1
      { S7_Templates := "SrcType := DInt" } GT_Contact(in1 := "Avoid".Av_2to3.V_Busy, in2 := 0)
      I_Contact( "M_A_2to3_L2-L2_B1" )
      Move(in := 1, out1 => "Cnv2".Sect3.H.V_Busy)
   END_RUNG
   RUNG wire#w1
      Contact( "M_A_2to3_L2-L2_B1" )
      { S7_Templates := "SrcType := DInt" } GT_Contact(in1 := "Cnv2".Sect3.H.V_Busy, in2 := 0)
      P_Trig( "M_B2H_S3_2_Trig2" )
      Sub(in1 := "Cnv2".Sect3.H.V_Busy, in2 := 1, out => "Cnv2".Sect3.H.V_Busy)
   END_RUNG
   RUNG wire#w1
      { S7_Templates := "SrcType := DInt" } GE_Contact(in1 := "Cnv2".Sect3.H.V_NumOfBox, in2 := 1)
      R_Coil( "M_B2H_S3_1" )
   END_RUNG
   RUNG wire#w1
      { S7_Templates := "SrcType := DInt" } GT_Contact(in1 := "Cnv2".Sect3.H.I_RFID_1, in2 := 0)
      P_Trig( "M_B2H_S3_2_Trig3" )
      "Enqueue3"("Array" := "Avoid".Av_2to3.V_BoxQueue, Input := "Cnv2".Sect3.H.I_RFID_1, size := "Avoid".Av_2to3.V_NumOfBoxWaiting)
   END_RUNG
   // the same network as SCL:
   IF "M_B2H_S3_2" AND ("Avoid".Av_2to3.V_Busy > 0) AND NOT "M_A_2to3_L2-L2_B1" THEN
       "Cnv2".Sect3.H.V_Busy := 1;
   END_IF;
   #_w1 := "M_B2H_S3_2" AND "M_A_2to3_L2-L2_B1" AND ("Cnv2".Sect3.H.V_Busy > 0);
   #_w2 := #_w1 AND NOT "M_B2H_S3_2_Trig2";   // rising edge
   "M_B2H_S3_2_Trig2" := #_w1;
   IF #_w2 THEN "Cnv2".Sect3.H.V_Busy := "Cnv2".Sect3.H.V_Busy - 1; END_IF;
   IF "M_B2H_S3_2" AND ("Cnv2".Sect3.H.V_NumOfBox >= 1) THEN "M_B2H_S3_1" := FALSE; END_IF;
   #_w3 := "M_B2H_S3_2" AND ("Cnv2".Sect3.H.I_RFID_1 > 0);
   #_w4 := #_w3 AND NOT "M_B2H_S3_2_Trig3";   // rising edge
   "M_B2H_S3_2_Trig3" := #_w3;
   IF #_w4 THEN
       "Enqueue3"("Array" := "Avoid".Av_2to3.V_BoxQueue,
                  Input := "Cnv2".Sect3.H.I_RFID_1,
                  size := "Avoid".Av_2to3.V_NumOfBoxWaiting);
   END_IF;
END_REGION

REGION Network 153: Mode back sect 4 high input - activate
   RUNG wire#powerrail
      Contact( "M_UD_4_B_7" )
      { S7_Templates := "SrcType := DInt" } GT_Contact(in1 := "Cnv2".Sect4.H.I_RFID_2, in2 := 0)
      S_Coil( "M_B2H_S4_1" )
   END_RUNG
   // the same network as SCL:
   IF "M_UD_4_B_7" AND ("Cnv2".Sect4.H.I_RFID_2 > 0) THEN "M_B2H_S4_1" := TRUE; END_IF;
END_REGION

REGION Network 154: Mode back sect 4 high input
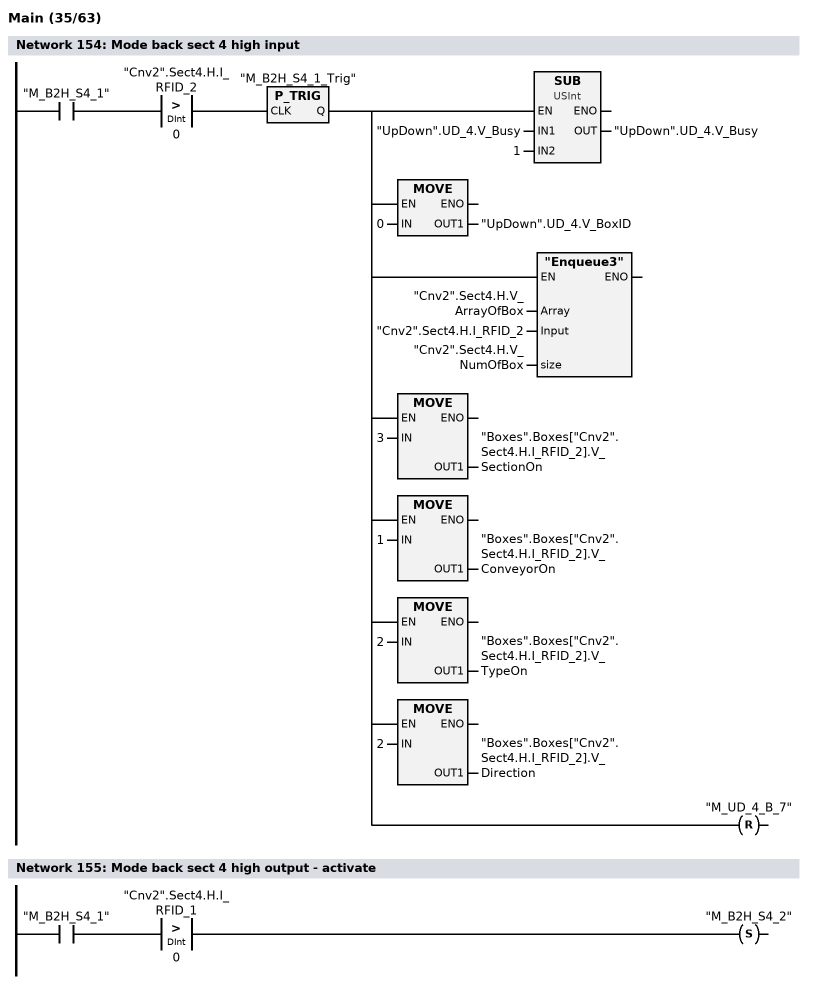
   RUNG wire#powerrail
      Contact( "M_B2H_S4_1" )
      { S7_Templates := "SrcType := DInt" } GT_Contact(in1 := "Cnv2".Sect4.H.I_RFID_2, in2 := 0)
      P_Trig( "M_B2H_S4_1_Trig" )
      wire#w1
      { S7_Templates := "SrcType := USInt" } Sub(in1 := "UpDown".UD_4.V_Busy, in2 := 1, out => "UpDown".UD_4.V_Busy)
   END_RUNG
   RUNG wire#w1
      Move(in := 0, out1 => "UpDown".UD_4.V_BoxID)
   END_RUNG
   RUNG wire#w1
      "Enqueue3"("Array" := "Cnv2".Sect4.H.V_ArrayOfBox, Input := "Cnv2".Sect4.H.I_RFID_2, size := "Cnv2".Sect4.H.V_NumOfBox)
   END_RUNG
   RUNG wire#w1
      Move(in := 3, out1 => "Boxes".Boxes["Cnv2".Sect4.H.I_RFID_2].V_SectionOn)
   END_RUNG
   RUNG wire#w1
      Move(in := 1, out1 => "Boxes".Boxes["Cnv2".Sect4.H.I_RFID_2].V_ConveyorOn)
   END_RUNG
   RUNG wire#w1
      Move(in := 2, out1 => "Boxes".Boxes["Cnv2".Sect4.H.I_RFID_2].V_TypeOn)
   END_RUNG
   RUNG wire#w1
      Move(in := 2, out1 => "Boxes".Boxes["Cnv2".Sect4.H.I_RFID_2].V_Direction)
   END_RUNG
   RUNG wire#w1
      R_Coil( "M_UD_4_B_7" )
   END_RUNG
   // the same network as SCL:
   #_w1 := "M_B2H_S4_1" AND ("Cnv2".Sect4.H.I_RFID_2 > 0);
   #_w2 := #_w1 AND NOT "M_B2H_S4_1_Trig";   // rising edge
   "M_B2H_S4_1_Trig" := #_w1;
   IF #_w2 THEN
       "UpDown".UD_4.V_Busy := "UpDown".UD_4.V_Busy - 1;
       "UpDown".UD_4.V_BoxID := 0;
       "Enqueue3"("Array" := "Cnv2".Sect4.H.V_ArrayOfBox,
                  Input := "Cnv2".Sect4.H.I_RFID_2,
                  size := "Cnv2".Sect4.H.V_NumOfBox);
       "Boxes".Boxes["Cnv2".Sect4.H.I_RFID_2].V_SectionOn := 3;
       "Boxes".Boxes["Cnv2".Sect4.H.I_RFID_2].V_ConveyorOn := 1;
       "Boxes".Boxes["Cnv2".Sect4.H.I_RFID_2].V_TypeOn := 2;
       "Boxes".Boxes["Cnv2".Sect4.H.I_RFID_2].V_Direction := 2;
       "M_UD_4_B_7" := FALSE;
   END_IF;
END_REGION

REGION Network 155: Mode back sect 4 high output - activate
   RUNG wire#powerrail
      Contact( "M_B2H_S4_1" )
      { S7_Templates := "SrcType := DInt" } GT_Contact(in1 := "Cnv2".Sect4.H.I_RFID_1, in2 := 0)
      S_Coil( "M_B2H_S4_2" )
   END_RUNG
   // the same network as SCL:
   IF "M_B2H_S4_1" AND ("Cnv2".Sect4.H.I_RFID_1 > 0) THEN "M_B2H_S4_2" := TRUE; END_IF;
END_REGION

REGION Network 156: Mode back sect 4 high output
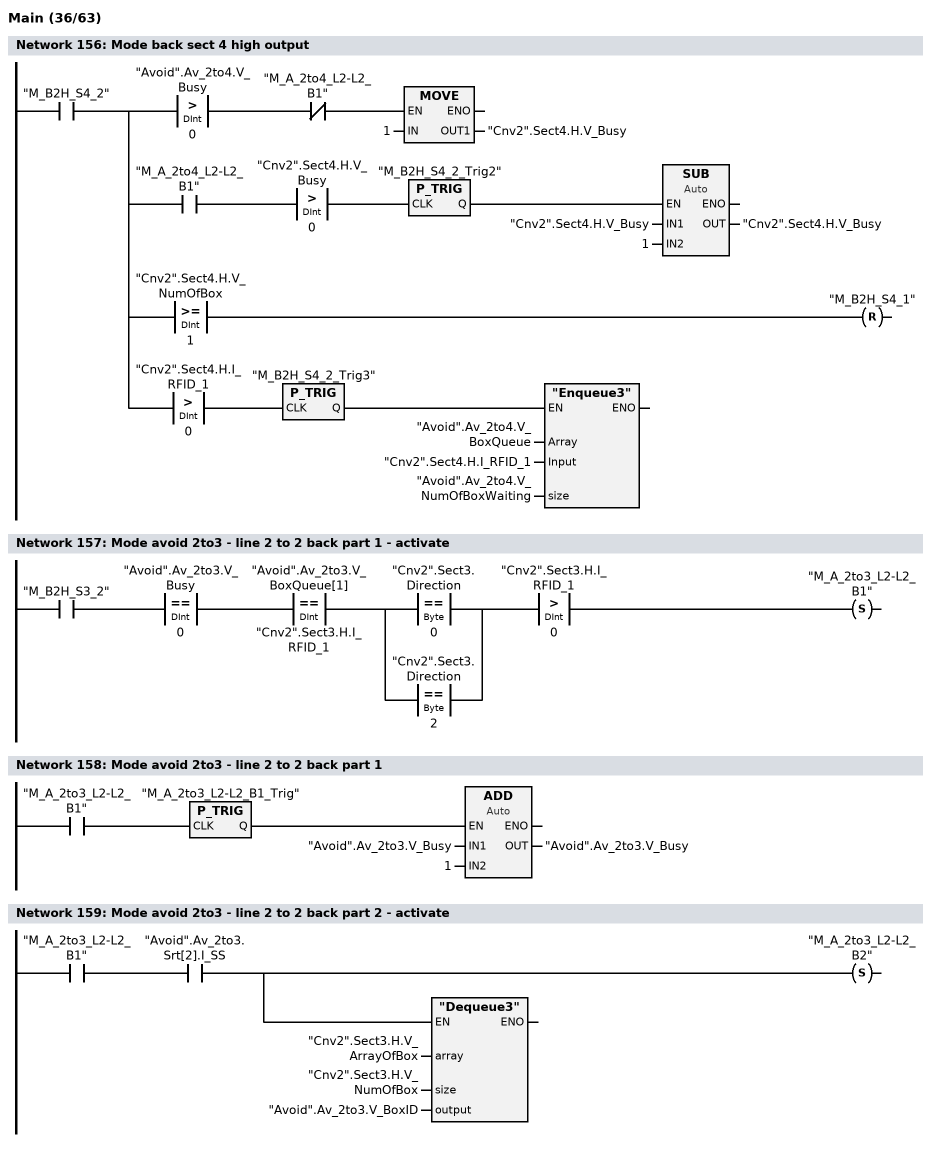
   RUNG wire#powerrail
      Contact( "M_B2H_S4_2" )
      wire#w1
      { S7_Templates := "SrcType := DInt" } GT_Contact(in1 := "Avoid".Av_2to4.V_Busy, in2 := 0)
      I_Contact( "M_A_2to4_L2-L2_B1" )
      Move(in := 1, out1 => "Cnv2".Sect4.H.V_Busy)
   END_RUNG
   RUNG wire#w1
      Contact( "M_A_2to4_L2-L2_B1" )
      { S7_Templates := "SrcType := DInt" } GT_Contact(in1 := "Cnv2".Sect4.H.V_Busy, in2 := 0)
      P_Trig( "M_B2H_S4_2_Trig2" )
      Sub(in1 := "Cnv2".Sect4.H.V_Busy, in2 := 1, out => "Cnv2".Sect4.H.V_Busy)
   END_RUNG
   RUNG wire#w1
      { S7_Templates := "SrcType := DInt" } GE_Contact(in1 := "Cnv2".Sect4.H.V_NumOfBox, in2 := 1)
      R_Coil( "M_B2H_S4_1" )
   END_RUNG
   RUNG wire#w1
      { S7_Templates := "SrcType := DInt" } GT_Contact(in1 := "Cnv2".Sect4.H.I_RFID_1, in2 := 0)
      P_Trig( "M_B2H_S4_2_Trig3" )
      "Enqueue3"("Array" := "Avoid".Av_2to4.V_BoxQueue, Input := "Cnv2".Sect4.H.I_RFID_1, size := "Avoid".Av_2to4.V_NumOfBoxWaiting)
   END_RUNG
   // the same network as SCL:
   IF "M_B2H_S4_2" AND ("Avoid".Av_2to4.V_Busy > 0) AND NOT "M_A_2to4_L2-L2_B1" THEN
       "Cnv2".Sect4.H.V_Busy := 1;
   END_IF;
   #_w1 := "M_B2H_S4_2" AND "M_A_2to4_L2-L2_B1" AND ("Cnv2".Sect4.H.V_Busy > 0);
   #_w2 := #_w1 AND NOT "M_B2H_S4_2_Trig2";   // rising edge
   "M_B2H_S4_2_Trig2" := #_w1;
   IF #_w2 THEN "Cnv2".Sect4.H.V_Busy := "Cnv2".Sect4.H.V_Busy - 1; END_IF;
   IF "M_B2H_S4_2" AND ("Cnv2".Sect4.H.V_NumOfBox >= 1) THEN "M_B2H_S4_1" := FALSE; END_IF;
   #_w3 := "M_B2H_S4_2" AND ("Cnv2".Sect4.H.I_RFID_1 > 0);
   #_w4 := #_w3 AND NOT "M_B2H_S4_2_Trig3";   // rising edge
   "M_B2H_S4_2_Trig3" := #_w3;
   IF #_w4 THEN
       "Enqueue3"("Array" := "Avoid".Av_2to4.V_BoxQueue,
                  Input := "Cnv2".Sect4.H.I_RFID_1,
                  size := "Avoid".Av_2to4.V_NumOfBoxWaiting);
   END_IF;
END_REGION

REGION Network 157: Mode avoid 2to3 - line 2 to 2 back part 1 - activate
   RUNG wire#powerrail
      Contact( "M_B2H_S3_2" )
      { S7_Templates := "SrcType := DInt" } EQ_Contact(in1 := "Avoid".Av_2to3.V_Busy, in2 := 0)
      { S7_Templates := "SrcType := DInt" } EQ_Contact(in1 := "Avoid".Av_2to3.V_BoxQueue[1], in2 := "Cnv2".Sect3.H.I_RFID_1)
      wire#w1
      { S7_Templates := "SrcType := Byte" } EQ_Contact(in1 := "Cnv2".Sect3.Direction, in2 := 0)
      wire#w2
      { S7_Templates := "SrcType := DInt" } GT_Contact(in1 := "Cnv2".Sect3.H.I_RFID_1, in2 := 0)
      S_Coil( "M_A_2to3_L2-L2_B1" )
   END_RUNG
   RUNG wire#w1
      { S7_Templates := "SrcType := Byte" } EQ_Contact(in1 := "Cnv2".Sect3.Direction, in2 := 2)
   END_RUNG wire#w2
   // the same network as SCL:
   IF "M_B2H_S3_2" AND ("Avoid".Av_2to3.V_Busy = 0) AND ("Avoid".Av_2to3.V_BoxQueue[1] = "Cnv2".Sect3.H.I_RFID_1) AND (("Cnv2".Sect3.Direction = 0) OR ("Cnv2".Sect3.Direction = 2)) AND ("Cnv2".Sect3.H.I_RFID_1 > 0) THEN
       "M_A_2to3_L2-L2_B1" := TRUE;
   END_IF;
END_REGION

REGION Network 158: Mode avoid 2to3 - line 2 to 2 back part 1
   RUNG wire#powerrail
      Contact( "M_A_2to3_L2-L2_B1" )
      P_Trig( "M_A_2to3_L2-L2_B1_Trig" )
      Add(in1 := "Avoid".Av_2to3.V_Busy, in2 := 1, out => "Avoid".Av_2to3.V_Busy)
   END_RUNG
   // the same network as SCL:
   #_w1 := "M_A_2to3_L2-L2_B1" AND NOT "M_A_2to3_L2-L2_B1_Trig";   // rising edge
   "M_A_2to3_L2-L2_B1_Trig" := "M_A_2to3_L2-L2_B1";
   IF #_w1 THEN "Avoid".Av_2to3.V_Busy := "Avoid".Av_2to3.V_Busy + 1; END_IF;
END_REGION

REGION Network 159: Mode avoid 2to3 - line 2 to 2 back part 2 - activate
   RUNG wire#powerrail
      Contact( "M_A_2to3_L2-L2_B1" )
      Contact( "Avoid".Av_2to3.Srt[2].I_SS )
      wire#w1
      S_Coil( "M_A_2to3_L2-L2_B2" )
   END_RUNG
   RUNG wire#w1
      "Dequeue3"("array" := "Cnv2".Sect3.H.V_ArrayOfBox, size := "Cnv2".Sect3.H.V_NumOfBox, output := "Avoid".Av_2to3.V_BoxID)
   END_RUNG
   // the same network as SCL:
   IF "M_A_2to3_L2-L2_B1" AND "Avoid".Av_2to3.Srt[2].I_SS THEN
       "M_A_2to3_L2-L2_B2" := TRUE;
       "Dequeue3"("array" := "Cnv2".Sect3.H.V_ArrayOfBox,
                  size := "Cnv2".Sect3.H.V_NumOfBox,
                  output := "Avoid".Av_2to3.V_BoxID);
   END_IF;
END_REGION

REGION Network 160: Mode avoid 2to3 - line 2 to 2 back part 2
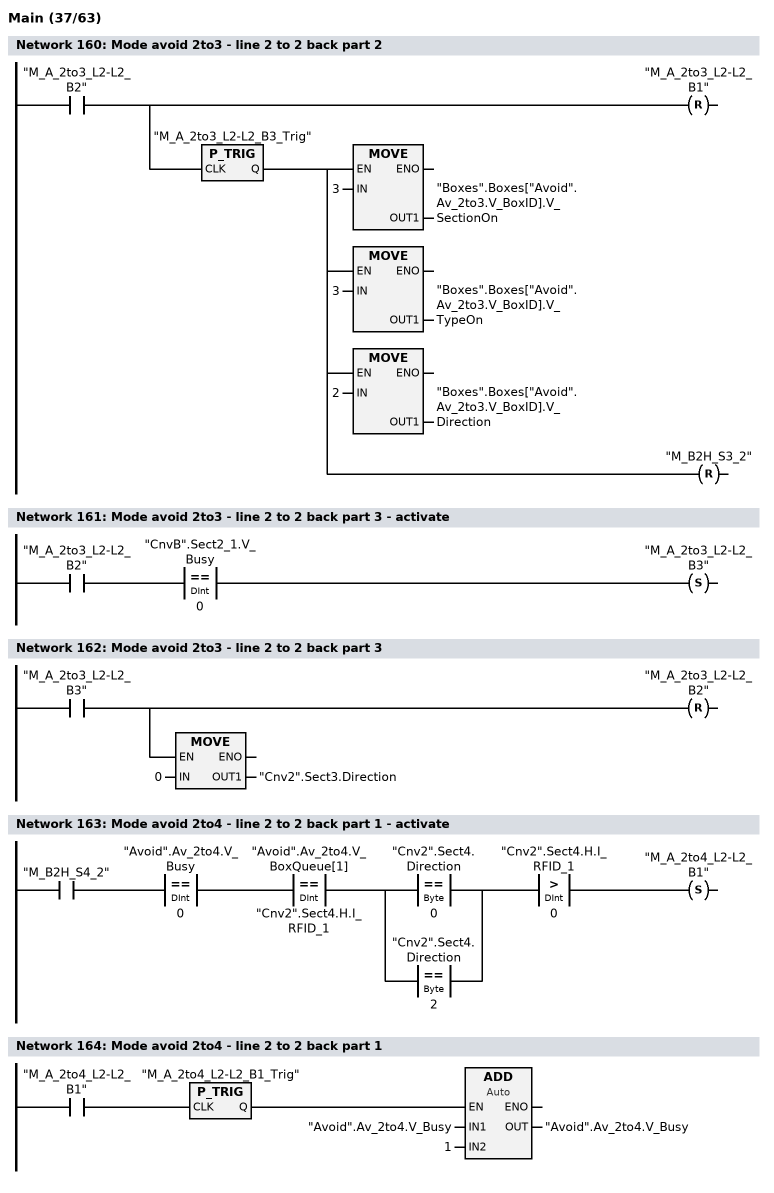
   RUNG wire#powerrail
      Contact( "M_A_2to3_L2-L2_B2" )
      wire#w1
      R_Coil( "M_A_2to3_L2-L2_B1" )
   END_RUNG
   RUNG wire#w1
      P_Trig( "M_A_2to3_L2-L2_B3_Trig" )
      wire#w2
      Move(in := 3, out1 => "Boxes".Boxes["Avoid".Av_2to3.V_BoxID].V_SectionOn)
   END_RUNG
   RUNG wire#w2
      Move(in := 3, out1 => "Boxes".Boxes["Avoid".Av_2to3.V_BoxID].V_TypeOn)
   END_RUNG
   RUNG wire#w2
      Move(in := 2, out1 => "Boxes".Boxes["Avoid".Av_2to3.V_BoxID].V_Direction)
   END_RUNG
   RUNG wire#w2
      R_Coil( "M_B2H_S3_2" )
   END_RUNG
   // the same network as SCL:
   IF "M_A_2to3_L2-L2_B2" THEN "M_A_2to3_L2-L2_B1" := FALSE; END_IF;
   #_w1 := "M_A_2to3_L2-L2_B2" AND NOT "M_A_2to3_L2-L2_B3_Trig";   // rising edge
   "M_A_2to3_L2-L2_B3_Trig" := "M_A_2to3_L2-L2_B2";
   IF #_w1 THEN
       "Boxes".Boxes["Avoid".Av_2to3.V_BoxID].V_SectionOn := 3;
       "Boxes".Boxes["Avoid".Av_2to3.V_BoxID].V_TypeOn := 3;
       "Boxes".Boxes["Avoid".Av_2to3.V_BoxID].V_Direction := 2;
       "M_B2H_S3_2" := FALSE;
   END_IF;
END_REGION

REGION Network 161: Mode avoid 2to3 - line 2 to 2 back part 3 - activate
   RUNG wire#powerrail
      Contact( "M_A_2to3_L2-L2_B2" )
      { S7_Templates := "SrcType := DInt" } EQ_Contact(in1 := "CnvB".Sect2_1.V_Busy, in2 := 0)
      S_Coil( "M_A_2to3_L2-L2_B3" )
   END_RUNG
   // the same network as SCL:
   IF "M_A_2to3_L2-L2_B2" AND ("CnvB".Sect2_1.V_Busy = 0) THEN "M_A_2to3_L2-L2_B3" := TRUE; END_IF;
END_REGION

REGION Network 162: Mode avoid 2to3 - line 2 to 2 back part 3
   RUNG wire#powerrail
      Contact( "M_A_2to3_L2-L2_B3" )
      wire#w1
      R_Coil( "M_A_2to3_L2-L2_B2" )
   END_RUNG
   RUNG wire#w1
      Move(in := 0, out1 => "Cnv2".Sect3.Direction)
   END_RUNG
   // the same network as SCL:
   IF "M_A_2to3_L2-L2_B3" THEN
       "M_A_2to3_L2-L2_B2" := FALSE;
       "Cnv2".Sect3.Direction := 0;
   END_IF;
END_REGION

REGION Network 163: Mode avoid 2to4 - line 2 to 2 back part 1 - activate
   RUNG wire#powerrail
      Contact( "M_B2H_S4_2" )
      { S7_Templates := "SrcType := DInt" } EQ_Contact(in1 := "Avoid".Av_2to4.V_Busy, in2 := 0)
      { S7_Templates := "SrcType := DInt" } EQ_Contact(in1 := "Avoid".Av_2to4.V_BoxQueue[1], in2 := "Cnv2".Sect4.H.I_RFID_1)
      wire#w1
      { S7_Templates := "SrcType := Byte" } EQ_Contact(in1 := "Cnv2".Sect4.Direction, in2 := 0)
      wire#w2
      { S7_Templates := "SrcType := DInt" } GT_Contact(in1 := "Cnv2".Sect4.H.I_RFID_1, in2 := 0)
      S_Coil( "M_A_2to4_L2-L2_B1" )
   END_RUNG
   RUNG wire#w1
      { S7_Templates := "SrcType := Byte" } EQ_Contact(in1 := "Cnv2".Sect4.Direction, in2 := 2)
   END_RUNG wire#w2
   // the same network as SCL:
   IF "M_B2H_S4_2" AND ("Avoid".Av_2to4.V_Busy = 0) AND ("Avoid".Av_2to4.V_BoxQueue[1] = "Cnv2".Sect4.H.I_RFID_1) AND (("Cnv2".Sect4.Direction = 0) OR ("Cnv2".Sect4.Direction = 2)) AND ("Cnv2".Sect4.H.I_RFID_1 > 0) THEN
       "M_A_2to4_L2-L2_B1" := TRUE;
   END_IF;
END_REGION

REGION Network 164: Mode avoid 2to4 - line 2 to 2 back part 1
   RUNG wire#powerrail
      Contact( "M_A_2to4_L2-L2_B1" )
      P_Trig( "M_A_2to4_L2-L2_B1_Trig" )
      Add(in1 := "Avoid".Av_2to4.V_Busy, in2 := 1, out => "Avoid".Av_2to4.V_Busy)
   END_RUNG
   // the same network as SCL:
   #_w1 := "M_A_2to4_L2-L2_B1" AND NOT "M_A_2to4_L2-L2_B1_Trig";   // rising edge
   "M_A_2to4_L2-L2_B1_Trig" := "M_A_2to4_L2-L2_B1";
   IF #_w1 THEN "Avoid".Av_2to4.V_Busy := "Avoid".Av_2to4.V_Busy + 1; END_IF;
END_REGION

REGION Network 165: Mode avoid 2to4 - line 2 to 2 back part 2 - activate
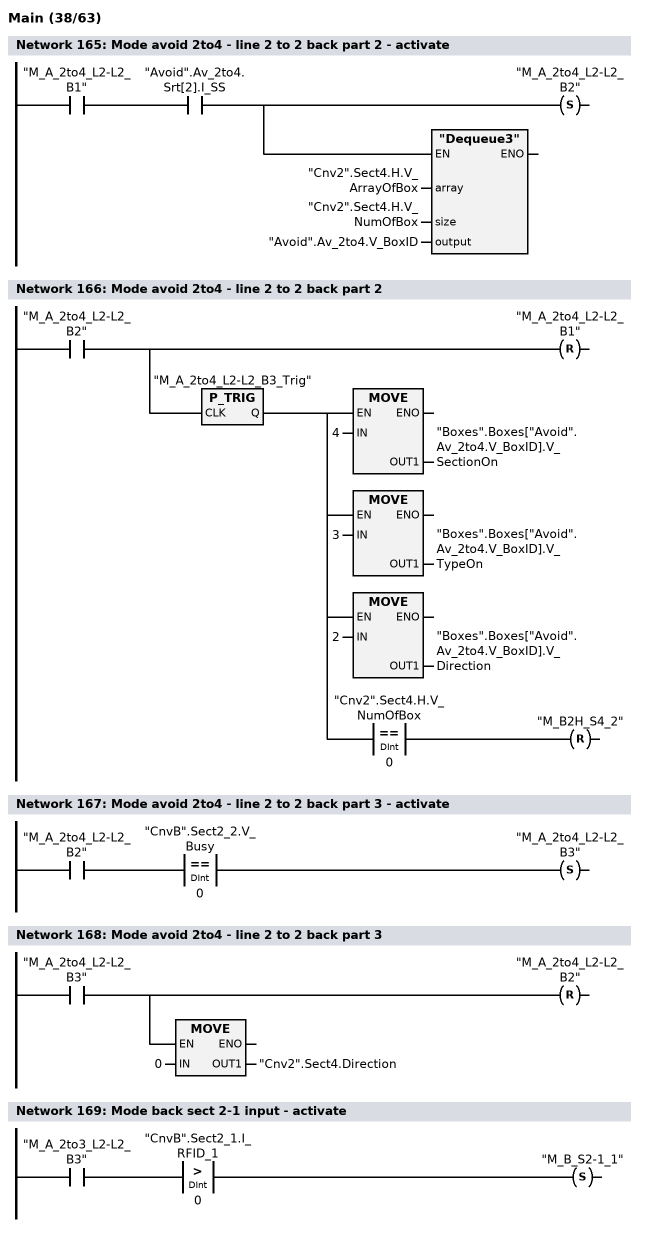
   RUNG wire#powerrail
      Contact( "M_A_2to4_L2-L2_B1" )
      Contact( "Avoid".Av_2to4.Srt[2].I_SS )
      wire#w1
      S_Coil( "M_A_2to4_L2-L2_B2" )
   END_RUNG
   RUNG wire#w1
      "Dequeue3"("array" := "Cnv2".Sect4.H.V_ArrayOfBox, size := "Cnv2".Sect4.H.V_NumOfBox, output := "Avoid".Av_2to4.V_BoxID)
   END_RUNG
   // the same network as SCL:
   IF "M_A_2to4_L2-L2_B1" AND "Avoid".Av_2to4.Srt[2].I_SS THEN
       "M_A_2to4_L2-L2_B2" := TRUE;
       "Dequeue3"("array" := "Cnv2".Sect4.H.V_ArrayOfBox,
                  size := "Cnv2".Sect4.H.V_NumOfBox,
                  output := "Avoid".Av_2to4.V_BoxID);
   END_IF;
END_REGION

REGION Network 166: Mode avoid 2to4 - line 2 to 2 back part 2
   RUNG wire#powerrail
      Contact( "M_A_2to4_L2-L2_B2" )
      wire#w1
      R_Coil( "M_A_2to4_L2-L2_B1" )
   END_RUNG
   RUNG wire#w1
      P_Trig( "M_A_2to4_L2-L2_B3_Trig" )
      wire#w2
      Move(in := 4, out1 => "Boxes".Boxes["Avoid".Av_2to4.V_BoxID].V_SectionOn)
   END_RUNG
   RUNG wire#w2
      Move(in := 3, out1 => "Boxes".Boxes["Avoid".Av_2to4.V_BoxID].V_TypeOn)
   END_RUNG
   RUNG wire#w2
      Move(in := 2, out1 => "Boxes".Boxes["Avoid".Av_2to4.V_BoxID].V_Direction)
   END_RUNG
   RUNG wire#w2
      { S7_Templates := "SrcType := DInt" } EQ_Contact(in1 := "Cnv2".Sect4.H.V_NumOfBox, in2 := 0)
      R_Coil( "M_B2H_S4_2" )
   END_RUNG
   // the same network as SCL:
   IF "M_A_2to4_L2-L2_B2" THEN "M_A_2to4_L2-L2_B1" := FALSE; END_IF;
   #_w1 := "M_A_2to4_L2-L2_B2" AND NOT "M_A_2to4_L2-L2_B3_Trig";   // rising edge
   "M_A_2to4_L2-L2_B3_Trig" := "M_A_2to4_L2-L2_B2";
   IF #_w1 THEN
       "Boxes".Boxes["Avoid".Av_2to4.V_BoxID].V_SectionOn := 4;
       "Boxes".Boxes["Avoid".Av_2to4.V_BoxID].V_TypeOn := 3;
       "Boxes".Boxes["Avoid".Av_2to4.V_BoxID].V_Direction := 2;
   END_IF;
   IF #_w1 AND ("Cnv2".Sect4.H.V_NumOfBox = 0) THEN "M_B2H_S4_2" := FALSE; END_IF;
END_REGION

REGION Network 167: Mode avoid 2to4 - line 2 to 2 back part 3 - activate
   RUNG wire#powerrail
      Contact( "M_A_2to4_L2-L2_B2" )
      { S7_Templates := "SrcType := DInt" } EQ_Contact(in1 := "CnvB".Sect2_2.V_Busy, in2 := 0)
      S_Coil( "M_A_2to4_L2-L2_B3" )
   END_RUNG
   // the same network as SCL:
   IF "M_A_2to4_L2-L2_B2" AND ("CnvB".Sect2_2.V_Busy = 0) THEN "M_A_2to4_L2-L2_B3" := TRUE; END_IF;
END_REGION

REGION Network 168: Mode avoid 2to4 - line 2 to 2 back part 3
   RUNG wire#powerrail
      Contact( "M_A_2to4_L2-L2_B3" )
      wire#w1
      R_Coil( "M_A_2to4_L2-L2_B2" )
   END_RUNG
   RUNG wire#w1
      Move(in := 0, out1 => "Cnv2".Sect4.Direction)
   END_RUNG
   // the same network as SCL:
   IF "M_A_2to4_L2-L2_B3" THEN
       "M_A_2to4_L2-L2_B2" := FALSE;
       "Cnv2".Sect4.Direction := 0;
   END_IF;
END_REGION

REGION Network 169: Mode back sect 2-1 input - activate
   RUNG wire#powerrail
      Contact( "M_A_2to3_L2-L2_B3" )
      { S7_Templates := "SrcType := DInt" } GT_Contact(in1 := "CnvB".Sect2_1.I_RFID_1, in2 := 0)
      S_Coil( "M_B_S2-1_1" )
   END_RUNG
   // the same network as SCL:
   IF "M_A_2to3_L2-L2_B3" AND ("CnvB".Sect2_1.I_RFID_1 > 0) THEN "M_B_S2-1_1" := TRUE; END_IF;
END_REGION

REGION Network 170: Mode back sect 2-1 input
